LIN {X 0,Y 133.955,Z 458.167,A -85,B 0,C 180,E1 -24920.946,E2 -24920.946} C_VEL
LIN {X 0,Y 133.688,Z 459.441,A -85,B 0,C 180,E1 -24923.966,E2 -24923.966} C_VEL
LIN {X 0,Y 133.69,Z 460.263,A -85,B 0,C 180,E1 -24927.209,E2 -24927.209} C_VEL
LIN {X 0,Y 133.919,Z 460.549,A -85,B 0,C 180,E1 -24930.002,E2 -24930.002} C_VEL
LIN {X 0,Y 133.701,Z 460.227,A -85,B 0,C 180,E1 -24933.015,E2 -24933.015} C_VEL
LIN {X 0,Y 133.689,Z 459.406,A -85,B 0,C 180,E1 -24936.037,E2 -24936.037} C_VEL
LIN {X 0,Y 133.956,Z 458.108,A -85,B 0,C 180,E1 -24939.057,E2 -24939.057} C_VEL
LIN {X 0,Y 134.932,Z 455.141,A -85,B 0,C 180,E1 -24943.557,E2 -24943.557} C_VEL
LIN {X 0,Y 136.058,Z 452.45,A -85,B 0,C 180,E1 -24946.507,E2 -24946.507} C_VEL
LIN {X 0,Y 138.397,Z 447.21,A -85,B 0,C 180,E1 -24950.824,E2 -24950.824} C_VEL
LIN {X 0,Y 141.592,Z 440.318,A -85,B 0,C 180,E1 -24954.956,E2 -24954.956} C_VEL
LIN {X 0,Y 144.781,Z 432.803,A -85,B 0,C 180,E1 -24958.249,E2 -24958.249} C_VEL
LIN {X 0,Y 145.009,Z 432.247,A -85,B 0,C 180,E1 -24958.457,E2 -24958.457} C_VEL
LIN {X 0,Y 146.09,Z 428.19,A -85,B 0,C 180,E1 -24960.037,E2 -24960.037} C_VEL
LIN {X 0,Y 146.273,Z 421.026,A -85,B 0,C 180,E1 -24962.704,E2 -24962.704} C_VEL
LIN {X 0,Y 146.437,Z 413.294,A -85,B 0,C 180,E1 -24965.152,E2 -24965.152} C_VEL
LIN {X 0,Y 147.423,Z 408.136,A -85,B 0,C 180,E1 -24966.312,E2 -24966.312} C_VEL
LIN {X 0,Y 150.465,Z 396.447,A -85,B 0,C 180,E1 -24968.09,E2 -24968.09} C_VEL
LIN {X 0,Y 152.454,Z 386.113,A -85,B 0,C 180,E1 -24969.14,E2 -24969.14} C_VEL
LIN {X 0,Y 153.592,Z 376.297,A -85,B 0,C 180,E1 -24969.839,E2 -24969.839} C_VEL
LIN {X 0,Y 154.357,Z 363.434,A -85,B 0,C 180,E1 -24970.454,E2 -24970.454} C_VEL
LIN {X 0,Y 152.82,Z 343.881,A -85,B 0,C 180,E1 -24972.135,E2 -24972.135} C_VEL
LIN {X 0,Y 148.055,Z 331.746,A -85,B 0,C 180,E1 -24974.6,E2 -24974.6} C_VEL
LIN {X 0,Y 143.112,Z 321.493,A -85,B 0,C 180,E1 -24977.289,E2 -24977.289} C_VEL
LIN {X 0,Y 138.714,Z 313.265,A -85,B 0,C 180,E1 -24979.904,E2 -24979.904} C_VEL
LIN {X 0,Y 135.903,Z 309.235,A -85,B 0,C 180,E1 -24981.643,E2 -24981.643} C_VEL
LIN {X 0,Y 133.491,Z 306.239,A -85,B 0,C 180,E1 -24983.212,E2 -24983.212} C_VEL
LIN {X 0,Y 132.602,Z 304.57,A -85,B 0,C 180,E1 -24983.869,E2 -24983.869} C_VEL
LIN {X 0,Y 130.375,Z 302.63,A -85,B 0,C 180,E1 -24985.393,E2 -24985.393} C_VEL
LIN {X 0,Y 129.129,Z 300.08,A -85,B 0,C 180,E1 -24986.438,E2 -24986.438} C_VEL
LIN {X 0,Y 128.983,Z 299.233,A -85,B 0,C 180,E1 -24986.69,E2 -24986.69} C_VEL
LIN {X 0,Y 128.983,Z 299.231,A -85,B 0,C 180,E1 -24990.672,E2 -24990.672} C_VEL
LIN {X 0,Y 129.069,Z 299.222,A -85,B 0,C 180,E1 -24997.774,E2 -24997.774} C_VEL
LIN {X 0,Y 129.147,Z 299.205,A -85,B 0,C 180,E1 -25004.211,E2 -25004.211} C_VEL
LIN {X 0,Y 129.346,Z 299.177,A -85,B 0,C 180,E1 -25007.974,E2 -25007.974} C_VEL
LIN {X 0,Y 129.462,Z 299.131,A -85,B 0,C 180,E1 -25010.628,E2 -25010.628} C_VEL
LIN {X 0,Y 130.069,Z 299.082,A -85,B 0,C 180,E1 -25020,E2 -25020} C_VEL
LIN {X 0,Y 129.471,Z 299.171,A -85,B 0,C 180,E1 -25029.373,E2 -25029.373} C_VEL
LIN {X 0,Y 129.3,Z 299.165,A -85,B 0,C 180,E1 -25032.558,E2 -25032.558} C_VEL
LIN {X 0,Y 129.083,Z 299.212,A -85,B 0,C 180,E1 -25039.067,E2 -25039.067} C_VEL
LIN {X 0,Y 129.036,Z 299.216,A -85,B 0,C 180,E1 -25042.412,E2 -25042.412} C_VEL
LIN {X 0,Y 129.002,Z 299.223,A -85,B 0,C 180,E1 -25049.362,E2 -25049.362} C_VEL
LIN {X 0,Y 129.003,Z 299.198,A -85,B 0,C 180,E1 -25054.184,E2 -25054.184} C_VEL
LIN {X 0,Y 129.928,Z 301.964,A -85,B 0,C 180,E1 -25055.083,E2 -25055.083} C_VEL
LIN {X 0,Y 131.991,Z 304.22,A -85,B 0,C 180,E1 -25056.562,E2 -25056.562} C_VEL
LIN {X 0,Y 132.836,Z 304.916,A -85,B 0,C 180,E1 -25057.12,E2 -25057.12} C_VEL
LIN {X 0,Y 134.792,Z 308.132,A -85,B 0,C 180,E1 -25058.493,E2 -25058.493} C_VEL
LIN {X 0,Y 136.443,Z 309.987,A -85,B 0,C 180,E1 -25059.521,E2 -25059.521} C_VEL
LIN {X 0,Y 139.015,Z 313.601,A -85,B 0,C 180,E1 -25061.089,E2 -25061.089} C_VEL
LIN {X 0,Y 144.709,Z 322.224,A -85,B 0,C 180,E1 -25064.255,E2 -25064.255} C_VEL
LIN {X 0,Y 149.932,Z 331.119,A -85,B 0,C 180,E1 -25066.875,E2 -25066.875} C_VEL
LIN {X 0,Y 155.317,Z 341.866,A -85,B 0,C 180,E1 -25069.382,E2 -25069.382} C_VEL
LIN {X 0,Y 155.665,Z 342.647,A -85,B 0,C 180,E1 -25069.54,E2 -25069.54} C_VEL
LIN {X 0,Y 154.337,Z 363.927,A -85,B 0,C 180,E1 -25070.495,E2 -25070.495} C_VEL
LIN {X 0,Y 153.217,Z 374.014,A -85,B 0,C 180,E1 -25071.268,E2 -25071.268} C_VEL
LIN {X 0,Y 151.609,Z 384.894,A -85,B 0,C 180,E1 -25072.59,E2 -25072.59} C_VEL
LIN {X 0,Y 149.044,Z 395.291,A -85,B 0,C 180,E1 -25074.299,E2 -25074.299} C_VEL
LIN {X 0,Y 146.437,Z 403.647,A -85,B 0,C 180,E1 -25076.086,E2 -25076.086} C_VEL
LIN {X 0,Y 143.646,Z 411.532,A -85,B 0,C 180,E1 -25078.266,E2 -25078.266} C_VEL
LIN {X 0,Y 141.558,Z 417.18,A -85,B 0,C 180,E1 -25080.231,E2 -25080.231} C_VEL
LIN {X 0,Y 138.779,Z 423.499,A -85,B 0,C 180,E1 -25082.884,E2 -25082.884} C_VEL
LIN {X 0,Y 136.313,Z 428.747,A -85,B 0,C 180,E1 -25085.639,E2 -25085.639} C_VEL
LIN {X 0,Y 134.031,Z 433.13,A -85,B 0,C 180,E1 -25088.465,E2 -25088.465} C_VEL
LIN {X 0,Y 131.319,Z 438.275,A -85,B 0,C 180,E1 -25092.88,E2 -25092.88} C_VEL
LIN {X 0,Y 129.865,Z 440.911,A -85,B 0,C 180,E1 -25095.903,E2 -25095.903} C_VEL
LIN {X 0,Y 128.338,Z 443.792,A -85,B 0,C 180,E1 -25100.543,E2 -25100.543} C_VEL
LIN {X 0,Y 127.603,Z 445.049,A -85,B 0,C 180,E1 -25103.674,E2 -25103.674} C_VEL
LIN {X 0,Y 127.149,Z 445.841,A -85,B 0,C 180,E1 -25106.83,E2 -25106.83} C_VEL
LIN {X 0,Y 127.002,Z 446.143,A -85,B 0,C 180,E1 -25109.998,E2 -25109.998} C_VEL
LIN {X 0,Y 127.144,Z 445.862,A -85,B 0,C 180,E1 -25113.167,E2 -25113.167} C_VEL
LIN {X 0,Y 127.58,Z 445.113,A -85,B 0,C 180,E1 -25116.324,E2 -25116.324} C_VEL
LIN {X 0,Y 128.518,Z 443.539,A -85,B 0,C 180,E1 -25120.155,E2 -25120.155} C_VEL
LIN {X 0,Y 129.861,Z 441.06,A -85,B 0,C 180,E1 -25124.094,E2 -25124.094} C_VEL
LIN {X 0,Y 131.287,Z 438.472,A -85,B 0,C 180,E1 -25127.121,E2 -25127.121} C_VEL
LIN {X 0,Y 133.978,Z 433.382,A -85,B 0,C 180,E1 -25131.541,E2 -25131.541} C_VEL
LIN {X 0,Y 136.782,Z 427.897,A -85,B 0,C 180,E1 -25135.079,E2 -25135.079} C_VEL
LIN {X 0,Y 140.081,Z 420.989,A -85,B 0,C 180,E1 -25138.463,E2 -25138.463} C_VEL
LIN {X 0,Y 143.2,Z 413.068,A -85,B 0,C 180,E1 -25141.428,E2 -25141.428} C_VEL
LIN {X 0,Y 146.001,Z 405.5,A -85,B 0,C 180,E1 -25143.61,E2 -25143.61} C_VEL
LIN {X 0,Y 148.554,Z 397.558,A -85,B 0,C 180,E1 -25145.416,E2 -25145.416} C_VEL
LIN {X 0,Y 150.694,Z 389.348,A -85,B 0,C 180,E1 -25146.901,E2 -25146.901} C_VEL
LIN {X 0,Y 152.252,Z 381.809,A -85,B 0,C 180,E1 -25147.985,E2 -25147.985} C_VEL
LIN {X 0,Y 153.626,Z 372.764,A -85,B 0,C 180,E1 -25148.981,E2 -25148.981} C_VEL
LIN {X 0,Y 154.497,Z 363.901,A -85,B 0,C 180,E1 -25149.672,E2 -25149.672} C_VEL
LIN {X 0,Y 155.859,Z 342.918,A -85,B 0,C 180,E1 -25150.597,E2 -25150.597} C_VEL
LIN {X 0,Y 150.73,Z 332.485,A -85,B 0,C 180,E1 -25152.978,E2 -25152.978} C_VEL
LIN {X 0,Y 145.136,Z 322.922,A -85,B 0,C 180,E1 -25155.765,E2 -25155.765} C_VEL
LIN {X 0,Y 140.991,Z 316.577,A -85,B 0,C 180,E1 -25158.021,E2 -25158.021} C_VEL
LIN {X 0,Y 138.32,Z 312.726,A -85,B 0,C 180,E1 -25159.585,E2 -25159.585} C_VEL
LIN {X 0,Y 135.823,Z 309.153,A -85,B 0,C 180,E1 -25161.152,E2 -25161.152} C_VEL
LIN {X 0,Y 133.437,Z 306.163,A -85,B 0,C 180,E1 -25162.721,E2 -25162.721} C_VEL
LIN {X 0,Y 132.55,Z 304.531,A -85,B 0,C 180,E1 -25163.381,E2 -25163.381} C_VEL
LIN {X 0,Y 130.335,Z 302.594,A -85,B 0,C 180,E1 -25164.913,E2 -25164.913} C_VEL
LIN {X 0,Y 129.126,Z 299.874,A -85,B 0,C 180,E1 -25165.962,E2 -25165.962} C_VEL
LIN {X 0,Y 128.982,Z 299.226,A -85,B 0,C 180,E1 -25166.275,E2 -25166.275} C_VEL
LIN {X 0,Y 129.014,Z 299.225,A -85,B 0,C 180,E1 -25170.641,E2 -25170.641} C_VEL
LIN {X 0,Y 128.999,Z 299.227,A -85,B 0,C 180,E1 -25174.16,E2 -25174.16} C_VEL
LIN {X 0,Y 129.066,Z 299.213,A -85,B 0,C 180,E1 -25177.769,E2 -25177.769} C_VEL
LIN {X 0,Y 129.14,Z 299.174,A -85,B 0,C 180,E1 -25184.21,E2 -25184.21} C_VEL
LIN {X 0,Y 129.339,Z 299.165,A -85,B 0,C 180,E1 -25187.973,E2 -25187.973} C_VEL
LIN {X 0,Y 129.464,Z 299.171,A -85,B 0,C 180,E1 -25190.627,E2 -25190.627} C_VEL
LIN {X 0,Y 130.062,Z 299.084,A -85,B 0,C 180,E1 -25200,E2 -25200} C_VEL
LIN {X 0,Y 129.464,Z 299.164,A -85,B 0,C 180,E1 -25209.372,E2 -25209.372} C_VEL
LIN {X 0,Y 129.293,Z 299.19,A -85,B 0,C 180,E1 -25212.558,E2 -25212.558} C_VEL
LIN {X 0,Y 129.076,Z 299.217,A -85,B 0,C 180,E1 -25219.068,E2 -25219.068} C_VEL
LIN {X 0,Y 129.03,Z 299.227,A -85,B 0,C 180,E1 -25222.412,E2 -25222.412} C_VEL
LIN {X 0,Y 128.995,Z 299.233,A -85,B 0,C 180,E1 -25229.363,E2 -25229.363} C_VEL
LIN {X 0,Y 128.964,Z 299.27,A -85,B 0,C 180,E1 -25233.139,E2 -25233.139} C_VEL
LIN {X 0,Y 129.82,Z 301.8,A -85,B 0,C 180,E1 -25233.949,E2 -25233.949} C_VEL
LIN {X 0,Y 131.932,Z 304.15,A -85,B 0,C 180,E1 -25235.486,E2 -25235.486} C_VEL
LIN {X 0,Y 132.916,Z 305.054,A -85,B 0,C 180,E1 -25236.149,E2 -25236.149} C_VEL
LIN {X 0,Y 134.987,Z 308.332,A -85,B 0,C 180,E1 -25237.598,E2 -25237.598} C_VEL
LIN {X 0,Y 136.451,Z 309.935,A -85,B 0,C 180,E1 -25238.511,E2 -25238.511} C_VEL
LIN {X 0,Y 139.616,Z 314.845,A -85,B 0,C 180,E1 -25240.475,E2 -25240.475} C_VEL
LIN {X 0,Y 144.191,Z 323.442,A -85,B 0,C 180,E1 -25243.148,E2 -25243.148} C_VEL
LIN {X 0,Y 149.027,Z 333.816,A -85,B 0,C 180,E1 -25245.756,E2 -25245.756} C_VEL
LIN {X 0,Y 153.092,Z 344.587,A -85,B 0,C 180,E1 -25247.869,E2 -25247.869} C_VEL
LIN {X 0,Y 154.559,Z 365.309,A -85,B 0,C 180,E1 -25249.596,E2 -25249.596} C_VEL
LIN {X 0,Y 153.372,Z 380.616,A -85,B 0,C 180,E1 -25250.333,E2 -25250.333} C_VEL
LIN {X 0,Y 151.602,Z 391.787,A -85,B 0,C 180,E1 -25251.311,E2 -25251.311} C_VEL
LIN {X 0,Y 149.671,Z 400.473,A -85,B 0,C 180,E1 -25252.381,E2 -25252.381} C_VEL
LIN {X 0,Y 147.268,Z 409.143,A -85,B 0,C 180,E1 -25253.805,E2 -25253.805} C_VEL
LIN {X 0,Y 144.547,Z 417.44,A -85,B 0,C 180,E1 -25255.586,E2 -25255.586} C_VEL
LIN {X 0,Y 141.851,Z 424.645,A -85,B 0,C 180,E1 -25257.553,E2 -25257.553} C_VEL
LIN {X 0,Y 138.564,Z 432.657,A -85,B 0,C 180,E1 -25260.364,E2 -25260.364} C_VEL
LIN {X 0,Y 135.155,Z 440.129,A -85,B 0,C 180,E1 -25263.771,E2 -25263.771} C_VEL
LIN {X 0,Y 132.3,Z 445.995,A -85,B 0,C 180,E1 -25267.35,E2 -25267.35} C_VEL
LIN {X 0,Y 129.937,Z 450.626,A -85,B 0,C 180,E1 -25271.065,E2 -25271.065} C_VEL
LIN {X 0,Y 128.595,Z 453.651,A -85,B 0,C 180,E1 -25274.143,E2 -25274.143} C_VEL
LIN {X 0,Y 127.585,Z 456.005,A -85,B 0,C 180,E1 -25277.273,E2 -25277.273} C_VEL
LIN {X 0,Y 126.927,Z 457.774,A -85,B 0,C 180,E1 -25280.44,E2 -25280.44} C_VEL
LIN {X 0,Y 126.626,Z 459.049,A -85,B 0,C 180,E1 -25283.628,E2 -25283.628} C_VEL
LIN {X 0,Y 126.633,Z 459.91,A -85,B 0,C 180,E1 -25287.404,E2 -25287.404} C_VEL
LIN {X 0,Y 126.82,Z 460.157,A -85,B 0,C 180,E1 -25290.002,E2 -25290.002} C_VEL
LIN {X 0,Y 126.615,Z 459.835,A -85,B 0,C 180,E1 -25293.184,E2 -25293.184} C_VEL
LIN {X 0,Y 126.627,Z 459.013,A -85,B 0,C 180,E1 -25296.375,E2 -25296.375} C_VEL
LIN {X 0,Y 126.928,Z 457.715,A -85,B 0,C 180,E1 -25299.563,E2 -25299.563} C_VEL
LIN {X 0,Y 128.02,Z 454.747,A -85,B 0,C 180,E1 -25304.304,E2 -25304.304} C_VEL
LIN {X 0,Y 129.227,Z 452.054,A -85,B 0,C 180,E1 -25307.406,E2 -25307.406} C_VEL
LIN {X 0,Y 131.785,Z 446.817,A -85,B 0,C 180,E1 -25311.921,E2 -25311.921} C_VEL
LIN {X 0,Y 135.145,Z 439.921,A -85,B 0,C 180,E1 -25316.235,E2 -25316.235} C_VEL
LIN {X 0,Y 138.589,Z 432.366,A -85,B 0,C 180,E1 -25319.655,E2 -25319.655} C_VEL
LIN {X 0,Y 141.661,Z 425.004,A -85,B 0,C 180,E1 -25322.232,E2 -25322.232} C_VEL
LIN {X 0,Y 144.427,Z 417.444,A -85,B 0,C 180,E1 -25324.325,E2 -25324.325} C_VEL
LIN {X 0,Y 147.255,Z 408.695,A -85,B 0,C 180,E1 -25326.202,E2 -25326.202} C_VEL
LIN {X 0,Y 147.423,Z 408.136,A -85,B 0,C 180,E1 -25326.312,E2 -25326.312} C_VEL
LIN {X 0,Y 148.397,Z 402.979,A -85,B 0,C 180,E1 -25327.382,E2 -25327.382} C_VEL
LIN {X 0,Y 148.347,Z 394.3,A -85,B 0,C 180,E1 -25329.252,E2 -25329.252} C_VEL
LIN {X 0,Y 147.785,Z 385.247,A -85,B 0,C 180,E1 -25330.819,E2 -25330.819} C_VEL
LIN {X 0,Y 147.904,Z 379.504,A -85,B 0,C 180,E1 -25331.386,E2 -25331.386} C_VEL
LIN {X 0,Y 148.981,Z 364.614,A -85,B 0,C 180,E1 -25332.14,E2 -25332.14} C_VEL
LIN {X 0,Y 147.735,Z 346.63,A -85,B 0,C 180,E1 -25333.739,E2 -25333.739} C_VEL
LIN {X 0,Y 143.311,Z 335.144,A -85,B 0,C 180,E1 -25336.234,E2 -25336.234} C_VEL
LIN {X 0,Y 138.463,Z 324.854,A -85,B 0,C 180,E1 -25339.125,E2 -25339.125} C_VEL
LIN {X 0,Y 134.783,Z 318.011,A -85,B 0,C 180,E1 -25341.505,E2 -25341.505} C_VEL
LIN {X 0,Y 132.341,Z 314.562,A -85,B 0,C 180,E1 -25343.136,E2 -25343.136} C_VEL
LIN {X 0,Y 130.013,Z 311.221,A -85,B 0,C 180,E1 -25344.815,E2 -25344.815} C_VEL
LIN {X 0,Y 126.908,Z 307.447,A -85,B 0,C 180,E1 -25347.203,E2 -25347.203} C_VEL
LIN {X 0,Y 126.017,Z 305.712,A -85,B 0,C 180,E1 -25348.007,E2 -25348.007} C_VEL
LIN {X 0,Y 123.536,Z 303.83,A -85,B 0,C 180,E1 -25350.079,E2 -25350.079} C_VEL
LIN {X 0,Y 122.11,Z 301.179,A -85,B 0,C 180,E1 -25351.559,E2 -25351.559} C_VEL
LIN {X 0,Y 121.88,Z 300.112,A -85,B 0,C 180,E1 -25351.942,E2 -25351.942} C_VEL
LIN {X 0,Y 121.981,Z 300.104,A -85,B 0,C 180,E1 -25357.202,E2 -25357.202} C_VEL
LIN {X 0,Y 122.06,Z 300.089,A -85,B 0,C 180,E1 -25363.269,E2 -25363.269} C_VEL
LIN {X 0,Y 122.289,Z 300.058,A -85,B 0,C 180,E1 -25367.694,E2 -25367.694} C_VEL
LIN {X 0,Y 122.391,Z 300.014,A -85,B 0,C 180,E1 -25370.081,E2 -25370.081} C_VEL
LIN {X 0,Y 122.558,Z 300.027,A -85,B 0,C 180,E1 -25376.713,E2 -25376.713} C_VEL
LIN {X 0,Y 123.022,Z 299.958,A -85,B 0,C 180,E1 -25380,E2 -25380} C_VEL
LIN {X 0,Y 122.391,Z 300.026,A -85,B 0,C 180,E1 -25386.889,E2 -25386.889} C_VEL
LIN {X 0,Y 122.29,Z 300.039,A -85,B 0,C 180,E1 -25392.308,E2 -25392.308} C_VEL
LIN {X 0,Y 122.06,Z 300.056,A -85,B 0,C 180,E1 -25396.732,E2 -25396.732} C_VEL
LIN {X 0,Y 121.981,Z 300.094,A -85,B 0,C 180,E1 -25402.799,E2 -25402.799} C_VEL
LIN {X 0,Y 121.959,Z 300.136,A -85,B 0,C 180,E1 -25409.009,E2 -25409.009} C_VEL
LIN {X 0,Y 122.813,Z 302.78,A -85,B 0,C 180,E1 -25410.039,E2 -25410.039} C_VEL
LIN {X 0,Y 124.819,Z 305.005,A -85,B 0,C 180,E1 -25411.862,E2 -25411.862} C_VEL
LIN {X 0,Y 126.222,Z 306.072,A -85,B 0,C 180,E1 -25412.999,E2 -25412.999} C_VEL
LIN {X 0,Y 128.002,Z 309.087,A -85,B 0,C 180,E1 -25414.521,E2 -25414.521} C_VEL
LIN {X 0,Y 129.971,Z 311.162,A -85,B 0,C 180,E1 -25415.975,E2 -25415.975} C_VEL
LIN {X 0,Y 132.546,Z 314.779,A -85,B 0,C 180,E1 -25417.822,E2 -25417.822} C_VEL
LIN {X 0,Y 138.419,Z 323.322,A -85,B 0,C 180,E1 -25421.558,E2 -25421.558} C_VEL
LIN {X 0,Y 144.642,Z 333.733,A -85,B 0,C 180,E1 -25425.03,E2 -25425.03} C_VEL
LIN {X 0,Y 150.226,Z 344.979,A -85,B 0,C 180,E1 -25427.868,E2 -25427.868} C_VEL
LIN {X 0,Y 148.944,Z 364.375,A -85,B 0,C 180,E1 -25428.766,E2 -25428.766} C_VEL
LIN {X 0,Y 147.653,Z 375.081,A -85,B 0,C 180,E1 -25429.603,E2 -25429.603} C_VEL
LIN {X 0,Y 145.627,Z 386.917,A -85,B 0,C 180,E1 -25431.141,E2 -25431.141} C_VEL
LIN {X 0,Y 143.358,Z 395.687,A -85,B 0,C 180,E1 -25432.649,E2 -25432.649} C_VEL
LIN {X 0,Y 140.613,Z 404.043,A -85,B 0,C 180,E1 -25434.475,E2 -25434.475} C_VEL
LIN {X 0,Y 137.69,Z 411.925,A -85,B 0,C 180,E1 -25436.72,E2 -25436.72} C_VEL
LIN {X 0,Y 134.71,Z 419.265,A -85,B 0,C 180,E1 -25439.423,E2 -25439.423} C_VEL
LIN {X 0,Y 131.145,Z 426.708,A -85,B 0,C 180,E1 -25442.901,E2 -25442.901} C_VEL
LIN {X 0,Y 127.481,Z 433.522,A -85,B 0,C 180,E1 -25447.298,E2 -25447.298} C_VEL
LIN {X 0,Y 124.567,Z 438.667,A -85,B 0,C 180,E1 -25451.921,E2 -25451.921} C_VEL
LIN {X 0,Y 123.02,Z 441.303,A -85,B 0,C 180,E1 -25455.101,E2 -25455.101} C_VEL
LIN {X 0,Y 121.363,Z 444.183,A -85,B 0,C 180,E1 -25459.994,E2 -25459.994} C_VEL
LIN {X 0,Y 120.56,Z 445.441,A -85,B 0,C 180,E1 -25463.303,E2 -25463.303} C_VEL
LIN {X 0,Y 120.09,Z 446.232,A -85,B 0,C 180,E1 -25466.643,E2 -25466.643} C_VEL
LIN {X 0,Y 119.931,Z 446.533,A -85,B 0,C 180,E1 -25469.998,E2 -25469.998} C_VEL
LIN {X 0,Y 120.084,Z 446.253,A -85,B 0,C 180,E1 -25473.353,E2 -25473.353} C_VEL
LIN {X 0,Y 120.555,Z 445.503,A -85,B 0,C 180,E1 -25476.694,E2 -25476.694} C_VEL
LIN {X 0,Y 121.322,Z 444.289,A -85,B 0,C 180,E1 -25480.006,E2 -25480.006} C_VEL
LIN {X 0,Y 123.017,Z 441.45,A -85,B 0,C 180,E1 -25484.895,E2 -25484.895} C_VEL
LIN {X 0,Y 124.526,Z 438.863,A -85,B 0,C 180,E1 -25488.082,E2 -25488.082} C_VEL
LIN {X 0,Y 127.427,Z 433.771,A -85,B 0,C 180,E1 -25492.708,E2 -25492.708} C_VEL
LIN {X 0,Y 130.4,Z 428.286,A -85,B 0,C 180,E1 -25496.398,E2 -25496.398} C_VEL
LIN {X 0,Y 133.904,Z 421.377,A -85,B 0,C 180,E1 -25499.906,E2 -25499.906} C_VEL
LIN {X 0,Y 137.221,Z 413.455,A -85,B 0,C 180,E1 -25502.966,E2 -25502.966} C_VEL
LIN {X 0,Y 140.156,Z 405.887,A -85,B 0,C 180,E1 -25505.214,E2 -25505.214} C_VEL
LIN {X 0,Y 142.855,Z 397.943,A -85,B 0,C 180,E1 -25507.058,E2 -25507.058} C_VEL
LIN {X 0,Y 145.092,Z 389.733,A -85,B 0,C 180,E1 -25508.581,E2 -25508.581} C_VEL
LIN {X 0,Y 147.029,Z 380.751,A -85,B 0,C 180,E1 -25509.858,E2 -25509.858} C_VEL
LIN {X 0,Y 148.428,Z 371.27,A -85,B 0,C 180,E1 -25510.877,E2 -25510.877} C_VEL
LIN {X 0,Y 149.468,Z 360.824,A -85,B 0,C 180,E1 -25511.589,E2 -25511.589} C_VEL
LIN {X 0,Y 150.43,Z 345.249,A -85,B 0,C 180,E1 -25512.269,E2 -25512.269} C_VEL
LIN {X 0,Y 145.035,Z 334.384,A -85,B 0,C 180,E1 -25515.009,E2 -25515.009} C_VEL
LIN {X 0,Y 139.531,Z 325.12,A -85,B 0,C 180,E1 -25518.047,E2 -25518.047} C_VEL
LIN {X 0,Y 134.959,Z 318.208,A -85,B 0,C 180,E1 -25520.855,E2 -25520.855} C_VEL
LIN {X 0,Y 132.401,Z 314.611,A -85,B 0,C 180,E1 -25522.571,E2 -25522.571} C_VEL
LIN {X 0,Y 129.875,Z 310.919,A -85,B 0,C 180,E1 -25524.418,E2 -25524.418} C_VEL
LIN {X 0,Y 127.202,Z 307.944,A -85,B 0,C 180,E1 -25526.46,E2 -25526.46} C_VEL
LIN {X 0,Y 126.013,Z 305.69,A -85,B 0,C 180,E1 -25527.533,E2 -25527.533} C_VEL
LIN {X 0,Y 123.603,Z 303.9,A -85,B 0,C 180,E1 -25529.564,E2 -25529.564} C_VEL
LIN {X 0,Y 122.245,Z 301.395,A -85,B 0,C 180,E1 -25530.98,E2 -25530.98} C_VEL
LIN {X 0,Y 121.928,Z 300.101,A -85,B 0,C 180,E1 -25531.498,E2 -25531.498} C_VEL
LIN {X 0,Y 121.984,Z 300.094,A -85,B 0,C 180,E1 -25537.189,E2 -25537.189} C_VEL
LIN {X 0,Y 122.055,Z 300.061,A -85,B 0,C 180,E1 -25543.267,E2 -25543.267} C_VEL
LIN {X 0,Y 122.283,Z 300.038,A -85,B 0,C 180,E1 -25547.691,E2 -25547.691} C_VEL
LIN {X 0,Y 122.39,Z 300.051,A -85,B 0,C 180,E1 -25550.08,E2 -25550.08} C_VEL
LIN {X 0,Y 122.551,Z 299.988,A -85,B 0,C 180,E1 -25556.712,E2 -25556.712} C_VEL
LIN {X 0,Y 123.015,Z 299.961,A -85,B 0,C 180,E1 -25560,E2 -25560} C_VEL
LIN {X 0,Y 122.404,Z 300.046,A -85,B 0,C 180,E1 -25566.594,E2 -25566.594} C_VEL
LIN {X 0,Y 122.391,Z 300.042,A -85,B 0,C 180,E1 -25569.919,E2 -25569.919} C_VEL
LIN {X 0,Y 122.182,Z 300.078,A -85,B 0,C 180,E1 -25573.302,E2 -25573.302} C_VEL
LIN {X 0,Y 121.981,Z 300.097,A -85,B 0,C 180,E1 -25580.224,E2 -25580.224} C_VEL
LIN {X 0,Y 121.907,Z 300.109,A -85,B 0,C 180,E1 -25583.8,E2 -25583.8} C_VEL
LIN {X 0,Y 121.896,Z 300.161,A -85,B 0,C 180,E1 -25587.836,E2 -25587.836} C_VEL
LIN {X 0,Y 122.59,Z 302.371,A -85,B 0,C 180,E1 -25588.697,E2 -25588.697} C_VEL
LIN {X 0,Y 124.523,Z 304.801,A -85,B 0,C 180,E1 -25590.527,E2 -25590.527} C_VEL
LIN {X 0,Y 126.229,Z 306.082,A -85,B 0,C 180,E1 -25591.932,E2 -25591.932} C_VEL
LIN {X 0,Y 128.297,Z 309.395,A -85,B 0,C 180,E1 -25593.691,E2 -25593.691} C_VEL
LIN {X 0,Y 130.005,Z 311.16,A -85,B 0,C 180,E1 -25594.954,E2 -25594.954} C_VEL
LIN {X 0,Y 132.549,Z 314.771,A -85,B 0,C 180,E1 -25596.797,E2 -25596.797} C_VEL
LIN {X 0,Y 135.721,Z 319.451,A -85,B 0,C 180,E1 -25598.913,E2 -25598.913} C_VEL
LIN {X 0,Y 140.916,Z 329.78,A -85,B 0,C 180,E1 -25602.197,E2 -25602.197} C_VEL
LIN {X 0,Y 144.887,Z 338.802,A -85,B 0,C 180,E1 -25604.505,E2 -25604.505} C_VEL
LIN {X 0,Y 148.019,Z 347.59,A -85,B 0,C 180,E1 -25606.287,E2 -25606.287} C_VEL
LIN {X 0,Y 149.171,Z 365.627,A -85,B 0,C 180,E1 -25607.854,E2 -25607.854} C_VEL
LIN {X 0,Y 147.883,Z 380.953,A -85,B 0,C 180,E1 -25608.629,E2 -25608.629} C_VEL
LIN {X 0,Y 146.254,Z 390.916,A -85,B 0,C 180,E1 -25609.521,E2 -25609.521} C_VEL
LIN {X 0,Y 144.112,Z 400.087,A -85,B 0,C 180,E1 -25610.658,E2 -25610.658} C_VEL
LIN {X 0,Y 141.591,Z 408.755,A -85,B 0,C 180,E1 -25612.105,E2 -25612.105} C_VEL
LIN {X 0,Y 138.75,Z 417.052,A -85,B 0,C 180,E1 -25613.929,E2 -25613.929} C_VEL
LIN {X 0,Y 135.899,Z 424.256,A -85,B 0,C 180,E1 -25615.944,E2 -25615.944} C_VEL
LIN {X 0,Y 133.211,Z 430.555,A -85,B 0,C 180,E1 -25618.16,E2 -25618.16} C_VEL
LIN {X 0,Y 130.14,Z 436.89,A -85,B 0,C 180,E1 -25620.922,E2 -25620.922} C_VEL
LIN {X 0,Y 127.537,Z 442.167,A -85,B 0,C 180,E1 -25623.844,E2 -25623.844} C_VEL
LIN {X 0,Y 125.2,Z 446.568,A -85,B 0,C 180,E1 -25626.864,E2 -25626.864} C_VEL
LIN {X 0,Y 122.442,Z 451.773,A -85,B 0,C 180,E1 -25631.599,E2 -25631.599} C_VEL
LIN {X 0,Y 120.632,Z 455.611,A -85,B 0,C 180,E1 -25636.526,E2 -25636.526} C_VEL
LIN {X 0,Y 119.925,Z 457.383,A -85,B 0,C 180,E1 -25639.876,E2 -25639.876} C_VEL
LIN {X 0,Y 119.56,Z 458.657,A -85,B 0,C 180,E1 -25643.25,E2 -25643.25} C_VEL
LIN {X 0,Y 119.565,Z 459.573,A -85,B 0,C 180,E1 -25647.783,E2 -25647.783} C_VEL
LIN {X 0,Y 119.724,Z 459.766,A -85,B 0,C 180,E1 -25650.002,E2 -25650.002} C_VEL
LIN {X 0,Y 119.53,Z 459.443,A -85,B 0,C 180,E1 -25653.372,E2 -25653.372} C_VEL
LIN {X 0,Y 119.561,Z 458.62,A -85,B 0,C 180,E1 -25656.753,E2 -25656.753} C_VEL
LIN {X 0,Y 119.925,Z 457.322,A -85,B 0,C 180,E1 -25660.127,E2 -25660.127} C_VEL
LIN {X 0,Y 121.142,Z 454.353,A -85,B 0,C 180,E1 -25665.135,E2 -25665.135} C_VEL
LIN {X 0,Y 122.441,Z 451.659,A -85,B 0,C 180,E1 -25668.404,E2 -25668.404} C_VEL
LIN {X 0,Y 125.198,Z 446.421,A -85,B 0,C 180,E1 -25673.14,E2 -25673.14} C_VEL
LIN {X 0,Y 128.766,Z 439.524,A -85,B 0,C 180,E1 -25677.642,E2 -25677.642} C_VEL
LIN {X 0,Y 132.432,Z 432.013,A -85,B 0,C 180,E1 -25681.161,E2 -25681.161} C_VEL
LIN {X 0,Y 135.699,Z 424.546,A -85,B 0,C 180,E1 -25683.86,E2 -25683.86} C_VEL
LIN {X 0,Y 138.605,Z 417.047,A -85,B 0,C 180,E1 -25685.985,E2 -25685.985} C_VEL
LIN {X 0,Y 141.577,Z 408.298,A -85,B 0,C 180,E1 -25687.903,E2 -25687.903} C_VEL
LIN {X 0,Y 144.484,Z 398.024,A -85,B 0,C 180,E1 -25689.578,E2 -25689.578} C_VEL
LIN {X 0,Y 146.859,Z 386.769,A -85,B 0,C 180,E1 -25690.795,E2 -25690.795} C_VEL
LIN {X 0,Y 147.904,Z 379.504,A -85,B 0,C 180,E1 -25691.386,E2 -25691.386} C_VEL
LIN {X 0,Y 147.734,Z 375.689,A -85,B 0,C 180,E1 -25691.778,E2 -25691.778} C_VEL
LIN {X 0,Y 146.08,Z 369.808,A -85,B 0,C 180,E1 -25692.823,E2 -25692.823} C_VEL
LIN {X 0,Y 143.792,Z 362.747,A -85,B 0,C 180,E1 -25694.141,E2 -25694.141} C_VEL
LIN {X 0,Y 143.42,Z 360.197,A -85,B 0,C 180,E1 -25694.454,E2 -25694.454} C_VEL
LIN {X 0,Y 142.64,Z 349.116,A -85,B 0,C 180,E1 -25695.527,E2 -25695.527} C_VEL
LIN {X 0,Y 138.633,Z 338.403,A -85,B 0,C 180,E1 -25698.015,E2 -25698.015} C_VEL
LIN {X 0,Y 133.598,Z 327.483,A -85,B 0,C 180,E1 -25701.341,E2 -25701.341} C_VEL
LIN {X 0,Y 131.174,Z 323.051,A -85,B 0,C 180,E1 -25703.054,E2 -25703.054} C_VEL
LIN {X 0,Y 128.986,Z 319.915,A -85,B 0,C 180,E1 -25704.638,E2 -25704.638} C_VEL
LIN {X 0,Y 126.369,Z 316.216,A -85,B 0,C 180,E1 -25706.688,E2 -25706.688} C_VEL
LIN {X 0,Y 123.879,Z 312.802,A -85,B 0,C 180,E1 -25708.823,E2 -25708.823} C_VEL
LIN {X 0,Y 123.182,Z 311.874,A -85,B 0,C 180,E1 -25709.457,E2 -25709.457} C_VEL
LIN {X 0,Y 120.7,Z 309.314,A -85,B 0,C 180,E1 -25711.792,E2 -25711.792} C_VEL
LIN {X 0,Y 119.361,Z 306.746,A -85,B 0,C 180,E1 -25713.323,E2 -25713.323} C_VEL
LIN {X 0,Y 116.939,Z 305.194,A -85,B 0,C 180,E1 -25715.968,E2 -25715.968} C_VEL
LIN {X 0,Y 115.24,Z 302.41,A -85,B 0,C 180,E1 -25718.347,E2 -25718.347} C_VEL
LIN {X 0,Y 114.935,Z 300.977,A -85,B 0,C 180,E1 -25719.064,E2 -25719.064} C_VEL
LIN {X 0,Y 115.081,Z 300.962,A -85,B 0,C 180,E1 -25725.861,E2 -25725.861} C_VEL
LIN {X 0,Y 115.307,Z 300.901,A -85,B 0,C 180,E1 -25729.464,E2 -25729.464} C_VEL
LIN {X 0,Y 115.485,Z 300.905,A -85,B 0,C 180,E1 -25736.511,E2 -25736.511} C_VEL
LIN {X 0,Y 115.95,Z 300.837,A -85,B 0,C 180,E1 -25740,E2 -25740} C_VEL
LIN {X 0,Y 115.351,Z 300.905,A -85,B 0,C 180,E1 -25746.999,E2 -25746.999} C_VEL
LIN {X 0,Y 115.207,Z 300.916,A -85,B 0,C 180,E1 -25752.557,E2 -25752.557} C_VEL
LIN {X 0,Y 114.965,Z 300.948,A -85,B 0,C 180,E1 -25757.798,E2 -25757.798} C_VEL
LIN {X 0,Y 114.948,Z 301.145,A -85,B 0,C 180,E1 -25761.902,E2 -25761.902} C_VEL
LIN {X 0,Y 115.768,Z 303.607,A -85,B 0,C 180,E1 -25763.298,E2 -25763.298} C_VEL
LIN {X 0,Y 117.627,Z 305.827,A -85,B 0,C 180,E1 -25765.67,E2 -25765.67} C_VEL
LIN {X 0,Y 119.541,Z 306.998,A -85,B 0,C 180,E1 -25767.699,E2 -25767.699} C_VEL
LIN {X 0,Y 121.193,Z 309.986,A -85,B 0,C 180,E1 -25769.535,E2 -25769.535} C_VEL
LIN {X 0,Y 123.599,Z 312.317,A -85,B 0,C 180,E1 -25771.734,E2 -25771.734} C_VEL
LIN {X 0,Y 126.052,Z 315.92,A -85,B 0,C 180,E1 -25773.887,E2 -25773.887} C_VEL
LIN {X 0,Y 127.297,Z 317.475,A -85,B 0,C 180,E1 -25774.877,E2 -25774.877} C_VEL
LIN {X 0,Y 130.877,Z 322.682,A -85,B 0,C 180,E1 -25777.564,E2 -25777.564} C_VEL
LIN {X 0,Y 135.247,Z 329.262,A -85,B 0,C 180,E1 -25780.478,E2 -25780.478} C_VEL
LIN {X 0,Y 141.116,Z 339.48,A -85,B 0,C 180,E1 -25783.978,E2 -25783.978} C_VEL
LIN {X 0,Y 144.861,Z 347.157,A -85,B 0,C 180,E1 -25786.037,E2 -25786.037} C_VEL
LIN {X 0,Y 143.672,Z 365.156,A -85,B 0,C 180,E1 -25786.931,E2 -25786.931} C_VEL
LIN {X 0,Y 142.288,Z 375.959,A -85,B 0,C 180,E1 -25787.808,E2 -25787.808} C_VEL
LIN {X 0,Y 140.189,Z 387.313,A -85,B 0,C 180,E1 -25789.327,E2 -25789.327} C_VEL
LIN {X 0,Y 137.799,Z 396.082,A -85,B 0,C 180,E1 -25790.863,E2 -25790.863} C_VEL
LIN {X 0,Y 134.926,Z 404.437,A -85,B 0,C 180,E1 -25792.732,E2 -25792.732} C_VEL
LIN {X 0,Y 131.843,Z 412.319,A -85,B 0,C 180,E1 -25795.036,E2 -25795.036} C_VEL
LIN {X 0,Y 128.674,Z 419.658,A -85,B 0,C 180,E1 -25797.822,E2 -25797.822} C_VEL
LIN {X 0,Y 124.893,Z 427.101,A -85,B 0,C 180,E1 -25801.423,E2 -25801.423} C_VEL
LIN {X 0,Y 120.995,Z 433.914,A -85,B 0,C 180,E1 -25806.007,E2 -25806.007} C_VEL
LIN {X 0,Y 117.846,Z 439.06,A -85,B 0,C 180,E1 -25810.851,E2 -25810.851} C_VEL
LIN {X 0,Y 116.185,Z 441.695,A -85,B 0,C 180,E1 -25814.203,E2 -25814.203} C_VEL
LIN {X 0,Y 114.409,Z 444.574,A -85,B 0,C 180,E1 -25819.379,E2 -25819.379} C_VEL
LIN {X 0,Y 113.521,Z 445.833,A -85,B 0,C 180,E1 -25822.886,E2 -25822.886} C_VEL
LIN {X 0,Y 113.014,Z 446.623,A -85,B 0,C 180,E1 -25826.433,E2 -25826.433} C_VEL
LIN {X 0,Y 112.842,Z 446.924,A -85,B 0,C 180,E1 -25829.998,E2 -25829.998} C_VEL
LIN {X 0,Y 113.009,Z 446.644,A -85,B 0,C 180,E1 -25833.564,E2 -25833.564} C_VEL
LIN {X 0,Y 114.183,Z 444.965,A -85,B 0,C 180,E1 -25839.999,E2 -25839.999} C_VEL
LIN {X 0,Y 115.531,Z 442.977,A -85,B 0,C 180,E1 -25844.081,E2 -25844.081} C_VEL
LIN {X 0,Y 117.817,Z 439.252,A -85,B 0,C 180,E1 -25849.151,E2 -25849.151} C_VEL
LIN {X 0,Y 120.94,Z 434.159,A -85,B 0,C 180,E1 -25854.001,E2 -25854.001} C_VEL
LIN {X 0,Y 124.102,Z 428.675,A -85,B 0,C 180,E1 -25857.851,E2 -25857.851} C_VEL
LIN {X 0,Y 127.824,Z 421.765,A -85,B 0,C 180,E1 -25861.486,E2 -25861.486} C_VEL
LIN {X 0,Y 131.345,Z 413.842,A -85,B 0,C 180,E1 -25864.645,E2 -25864.645} C_VEL
LIN {X 0,Y 134.446,Z 406.273,A -85,B 0,C 180,E1 -25866.95,E2 -25866.95} C_VEL
LIN {X 0,Y 137.284,Z 398.328,A -85,B 0,C 180,E1 -25868.835,E2 -25868.835} C_VEL
LIN {X 0,Y 139.634,Z 390.117,A -85,B 0,C 180,E1 -25870.39,E2 -25870.39} C_VEL
LIN {X 0,Y 141.547,Z 381.691,A -85,B 0,C 180,E1 -25871.627,E2 -25871.627} C_VEL
LIN {X 0,Y 143.059,Z 372.284,A -85,B 0,C 180,E1 -25872.674,E2 -25872.674} C_VEL
LIN {X 0,Y 144.154,Z 362.075,A -85,B 0,C 180,E1 -25873.411,E2 -25873.411} C_VEL
LIN {X 0,Y 145.103,Z 347.554,A -85,B 0,C 180,E1 -25874.081,E2 -25874.081} C_VEL
LIN {X 0,Y 139.9,Z 337.191,A -85,B 0,C 180,E1 -25876.974,E2 -25876.974} C_VEL
LIN {X 0,Y 134.512,Z 327.997,A -85,B 0,C 180,E1 -25880.279,E2 -25880.279} C_VEL
LIN {X 0,Y 129.55,Z 320.545,A -85,B 0,C 180,E1 -25883.721,E2 -25883.721} C_VEL
LIN {X 0,Y 126.472,Z 316.291,A -85,B 0,C 180,E1 -25886.12,E2 -25886.12} C_VEL
LIN {X 0,Y 123.899,Z 312.838,A -85,B 0,C 180,E1 -25888.336,E2 -25888.336} C_VEL
LIN {X 0,Y 123.094,Z 311.764,A -85,B 0,C 180,E1 -25889.079,E2 -25889.079} C_VEL
LIN {X 0,Y 120.725,Z 309.331,A -85,B 0,C 180,E1 -25891.339,E2 -25891.339} C_VEL
LIN {X 0,Y 119.416,Z 306.759,A -85,B 0,C 180,E1 -25892.863,E2 -25892.863} C_VEL
LIN {X 0,Y 116.8,Z 305.022,A -85,B 0,C 180,E1 -25895.787,E2 -25895.787} C_VEL
LIN {X 0,Y 115.184,Z 302.228,A -85,B 0,C 180,E1 -25898.139,E2 -25898.139} C_VEL
LIN {X 0,Y 114.91,Z 300.979,A -85,B 0,C 180,E1 -25898.706,E2 -25898.706} C_VEL
LIN {X 0,Y 115.075,Z 300.922,A -85,B 0,C 180,E1 -25905.86,E2 -25905.86} C_VEL
LIN {X 0,Y 115.304,Z 300.929,A -85,B 0,C 180,E1 -25909.463,E2 -25909.463} C_VEL
LIN {X 0,Y 115.477,Z 300.867,A -85,B 0,C 180,E1 -25916.51,E2 -25916.51} C_VEL
LIN {X 0,Y 115.967,Z 300.836,A -85,B 0,C 180,E1 -25920,E2 -25920} C_VEL
LIN {X 0,Y 115.346,Z 300.927,A -85,B 0,C 180,E1 -25926.999,E2 -25926.999} C_VEL
LIN {X 0,Y 115.199,Z 300.945,A -85,B 0,C 180,E1 -25932.557,E2 -25932.557} C_VEL
LIN {X 0,Y 114.924,Z 300.981,A -85,B 0,C 180,E1 -25940.587,E2 -25940.587} C_VEL
LIN {X 0,Y 115.627,Z 303.334,A -85,B 0,C 180,E1 -25941.86,E2 -25941.86} C_VEL
LIN {X 0,Y 117.797,Z 305.94,A -85,B 0,C 180,E1 -25944.685,E2 -25944.685} C_VEL
LIN {X 0,Y 119.51,Z 306.978,A -85,B 0,C 180,E1 -25946.523,E2 -25946.523} C_VEL
LIN {X 0,Y 121.405,Z 310.236,A -85,B 0,C 180,E1 -25948.629,E2 -25948.629} C_VEL
LIN {X 0,Y 123.715,Z 312.447,A -85,B 0,C 180,E1 -25950.748,E2 -25950.748} C_VEL
LIN {X 0,Y 126.264,Z 316.094,A -85,B 0,C 180,E1 -25952.986,E2 -25952.986} C_VEL
LIN {X 0,Y 127.401,Z 317.564,A -85,B 0,C 180,E1 -25953.899,E2 -25953.899} C_VEL
LIN {X 0,Y 130.802,Z 322.448,A -85,B 0,C 180,E1 -25956.469,E2 -25956.469} C_VEL
LIN {X 0,Y 132.753,Z 325.754,A -85,B 0,C 180,E1 -25957.863,E2 -25957.863} C_VEL
LIN {X 0,Y 137.82,Z 336.297,A -85,B 0,C 180,E1 -25961.279,E2 -25961.279} C_VEL
LIN {X 0,Y 142.078,Z 347.187,A -85,B 0,C 180,E1 -25963.953,E2 -25963.953} C_VEL
LIN {X 0,Y 142.937,Z 349.704,A -85,B 0,C 180,E1 -25964.48,E2 -25964.48} C_VEL
LIN {X 0,Y 143.898,Z 366.473,A -85,B 0,C 180,E1 -25966.007,E2 -25966.007} C_VEL
LIN {X 0,Y 142.537,Z 381.175,A -85,B 0,C 180,E1 -25966.793,E2 -25966.793} C_VEL
LIN {X 0,Y 140.799,Z 391.081,A -85,B 0,C 180,E1 -25967.709,E2 -25967.709} C_VEL
LIN {X 0,Y 138.7,Z 399.702,A -85,B 0,C 180,E1 -25968.8,E2 -25968.8} C_VEL
LIN {X 0,Y 136.073,Z 408.368,A -85,B 0,C 180,E1 -25970.274,E2 -25970.274} C_VEL
LIN {X 0,Y 133.088,Z 416.66,A -85,B 0,C 180,E1 -25972.131,E2 -25972.131} C_VEL
LIN {X 0,Y 129.881,Z 424.303,A -85,B 0,C 180,E1 -25974.333,E2 -25974.333} C_VEL
LIN {X 0,Y 127.218,Z 430.164,A -85,B 0,C 180,E1 -25976.468,E2 -25976.468} C_VEL
LIN {X 0,Y 123.983,Z 436.5,A -85,B 0,C 180,E1 -25979.327,E2 -25979.327} C_VEL
LIN {X 0,Y 121.179,Z 441.775,A -85,B 0,C 180,E1 -25982.358,E2 -25982.358} C_VEL
LIN {X 0,Y 118.676,Z 446.176,A -85,B 0,C 180,E1 -25985.512,E2 -25985.512} C_VEL
LIN {X 0,Y 115.683,Z 451.38,A -85,B 0,C 180,E1 -25990.482,E2 -25990.482} C_VEL
LIN {X 0,Y 113.718,Z 455.219,A -85,B 0,C 180,E1 -25995.69,E2 -25995.69} C_VEL
LIN {X 0,Y 112.918,Z 456.99,A -85,B 0,C 180,E1 -25999.241,E2 -25999.241} C_VEL
LIN {X 0,Y 112.492,Z 458.264,A -85,B 0,C 180,E1 -26002.824,E2 -26002.824} C_VEL
LIN {X 0,Y 112.496,Z 459.245,A -85,B 0,C 180,E1 -26008.317,E2 -26008.317} C_VEL
LIN {X 0,Y 112.625,Z 459.374,A -85,B 0,C 180,E1 -26010.002,E2 -26010.002} C_VEL
LIN {X 0,Y 112.43,Z 459.05,A -85,B 0,C 180,E1 -26013.586,E2 -26013.586} C_VEL
LIN {X 0,Y 112.493,Z 458.227,A -85,B 0,C 180,E1 -26017.18,E2 -26017.18} C_VEL
LIN {X 0,Y 112.918,Z 456.928,A -85,B 0,C 180,E1 -26020.763,E2 -26020.763} C_VEL
LIN {X 0,Y 114.278,Z 453.959,A -85,B 0,C 180,E1 -26026.068,E2 -26026.068} C_VEL
LIN {X 0,Y 115.683,Z 451.264,A -85,B 0,C 180,E1 -26029.522,E2 -26029.522} C_VEL
LIN {X 0,Y 118.674,Z 446.026,A -85,B 0,C 180,E1 -26034.493,E2 -26034.493} C_VEL
LIN {X 0,Y 122.489,Z 439.128,A -85,B 0,C 180,E1 -26039.191,E2 -26039.191} C_VEL
LIN {X 0,Y 126.403,Z 431.617,A -85,B 0,C 180,E1 -26042.828,E2 -26042.828} C_VEL
LIN {X 0,Y 129.371,Z 425.254,A -85,B 0,C 180,E1 -26045.247,E2 -26045.247} C_VEL
LIN {X 0,Y 132.585,Z 417.515,A -85,B 0,C 180,E1 -26047.561,E2 -26047.561} C_VEL
LIN {X 0,Y 135.532,Z 409.405,A -85,B 0,C 180,E1 -26049.438,E2 -26049.438} C_VEL
LIN {X 0,Y 138.114,Z 400.993,A -85,B 0,C 180,E1 -26050.933,E2 -26050.933} C_VEL
LIN {X 0,Y 140.751,Z 390.755,A -85,B 0,C 180,E1 -26052.229,E2 -26052.229} C_VEL
LIN {X 0,Y 142.753,Z 377.869,A -85,B 0,C 180,E1 -26053.349,E2 -26053.349} C_VEL
LIN {X 0,Y 143.718,Z 365.727,A -85,B 0,C 180,E1 -26053.965,E2 -26053.965} C_VEL
LIN {X 0,Y 143.42,Z 360.197,A -85,B 0,C 180,E1 -26054.454,E2 -26054.454} C_VEL
LIN {X 0,Y 142.814,Z 356.518,A -85,B 0,C 180,E1 -26054.943,E2 -26054.943} C_VEL
LIN {X 0,Y 141.009,Z 351.55,A -85,B 0,C 180,E1 -26056.023,E2 -26056.023} C_VEL
LIN {X 0,Y 138.588,Z 347.192,A -85,B 0,C 180,E1 -26057.378,E2 -26057.378} C_VEL
LIN {X 0,Y 131.659,Z 336.057,A -85,B 0,C 180,E1 -26061.654,E2 -26061.654} C_VEL
LIN {X 0,Y 128.004,Z 328.578,A -85,B 0,C 180,E1 -26064.434,E2 -26064.434} C_VEL
LIN {X 0,Y 123.709,Z 322.226,A -85,B 0,C 180,E1 -26067.939,E2 -26067.939} C_VEL
LIN {X 0,Y 120.7,Z 318.081,A -85,B 0,C 180,E1 -26070.743,E2 -26070.743} C_VEL
LIN {X 0,Y 118.237,Z 315.167,A -85,B 0,C 180,E1 -26073.288,E2 -26073.288} C_VEL
LIN {X 0,Y 116.991,Z 313.196,A -85,B 0,C 180,E1 -26074.777,E2 -26074.777} C_VEL
LIN {X 0,Y 114.633,Z 311.102,A -85,B 0,C 180,E1 -26077.686,E2 -26077.686} C_VEL
LIN {X 0,Y 113.048,Z 307.984,A -85,B 0,C 180,E1 -26080.243,E2 -26080.243} C_VEL
LIN {X 0,Y 109.847,Z 305.752,A -85,B 0,C 180,E1 -26085.999,E2 -26085.999} C_VEL
LIN {X 0,Y 108.332,Z 302.362,A -85,B 0,C 180,E1 -26090.784,E2 -26090.784} C_VEL
LIN {X 0,Y 108.24,Z 301.766,A -85,B 0,C 180,E1 -26091.6,E2 -26091.6} C_VEL
LIN {X 0,Y 108.879,Z 301.714,A -85,B 0,C 180,E1 -26100,E2 -26100} C_VEL
LIN {X 0,Y 108.274,Z 301.956,A -85,B 0,C 180,E1 -26109.693,E2 -26109.693} C_VEL
LIN {X 0,Y 109.233,Z 304.862,A -85,B 0,C 180,E1 -26113.255,E2 -26113.255} C_VEL
LIN {X 0,Y 111.384,Z 307.086,A -85,B 0,C 180,E1 -26117.915,E2 -26117.915} C_VEL
LIN {X 0,Y 113.056,Z 307.967,A -85,B 0,C 180,E1 -26120.587,E2 -26120.587} C_VEL
LIN {X 0,Y 114.456,Z 310.937,A -85,B 0,C 180,E1 -26122.898,E2 -26122.898} C_VEL
LIN {X 0,Y 116.822,Z 313.11,A -85,B 0,C 180,E1 -26125.86,E2 -26125.86} C_VEL
LIN {X 0,Y 117.427,Z 313.692,A -85,B 0,C 180,E1 -26126.552,E2 -26126.552} C_VEL
LIN {X 0,Y 119.59,Z 317.015,A -85,B 0,C 180,E1 -26129.002,E2 -26129.002} C_VEL
LIN {X 0,Y 121.235,Z 318.774,A -85,B 0,C 180,E1 -26130.601,E2 -26130.601} C_VEL
LIN {X 0,Y 124.889,Z 324.01,A -85,B 0,C 180,E1 -26133.907,E2 -26133.907} C_VEL
LIN {X 0,Y 127.744,Z 328.263,A -85,B 0,C 180,E1 -26136.198,E2 -26136.198} C_VEL
LIN {X 0,Y 132.366,Z 335.601,A -85,B 0,C 180,E1 -26139.509,E2 -26139.509} C_VEL
LIN {X 0,Y 137.159,Z 344.369,A -85,B 0,C 180,E1 -26142.586,E2 -26142.586} C_VEL
LIN {X 0,Y 139.729,Z 349.792,A -85,B 0,C 180,E1 -26144.133,E2 -26144.133} C_VEL
LIN {X 0,Y 138.477,Z 366.762,A -85,B 0,C 180,E1 -26145.007,E2 -26145.007} C_VEL
LIN {X 0,Y 136.655,Z 379.188,A -85,B 0,C 180,E1 -26146.161,E2 -26146.161} C_VEL
LIN {X 0,Y 134.897,Z 387.71,A -85,B 0,C 180,E1 -26147.366,E2 -26147.366} C_VEL
LIN {X 0,Y 132.394,Z 396.477,A -85,B 0,C 180,E1 -26148.933,E2 -26148.933} C_VEL
LIN {X 0,Y 129.377,Z 404.831,A -85,B 0,C 180,E1 -26150.838,E2 -26150.838} C_VEL
LIN {X 0,Y 126.119,Z 412.712,A -85,B 0,C 180,E1 -26153.197,E2 -26153.197} C_VEL
LIN {X 0,Y 122.75,Z 420.051,A -85,B 0,C 180,E1 -26156.065,E2 -26156.065} C_VEL
LIN {X 0,Y 118.735,Z 427.494,A -85,B 0,C 180,E1 -26159.791,E2 -26159.791} C_VEL
LIN {X 0,Y 114.554,Z 434.307,A -85,B 0,C 180,E1 -26164.565,E2 -26164.565} C_VEL
LIN {X 0,Y 111.183,Z 439.452,A -85,B 0,C 180,E1 -26169.654,E2 -26169.654} C_VEL
LIN {X 0,Y 109.397,Z 442.086,A -85,B 0,C 180,E1 -26173.194,E2 -26173.194} C_VEL
LIN {X 0,Y 107.21,Z 445.327,A -85,B 0,C 180,E1 -26179.518,E2 -26179.518} C_VEL
LIN {X 0,Y 105.941,Z 447.015,A -85,B 0,C 180,E1 -26186.194,E2 -26186.194} C_VEL
LIN {X 0,Y 105.755,Z 447.316,A -85,B 0,C 180,E1 -26189.998,E2 -26189.998} C_VEL
LIN {X 0,Y 105.937,Z 447.035,A -85,B 0,C 180,E1 -26193.802,E2 -26193.802} C_VEL
LIN {X 0,Y 107.007,Z 445.671,A -85,B 0,C 180,E1 -26199.879,E2 -26199.879} C_VEL
LIN {X 0,Y 108.676,Z 443.367,A -85,B 0,C 180,E1 -26204.989,E2 -26204.989} C_VEL
LIN {X 0,Y 111.161,Z 439.641,A -85,B 0,C 180,E1 -26210.346,E2 -26210.346} C_VEL
LIN {X 0,Y 114.497,Z 434.549,A -85,B 0,C 180,E1 -26215.445,E2 -26215.445} C_VEL
LIN {X 0,Y 117.899,Z 429.063,A -85,B 0,C 180,E1 -26219.456,E2 -26219.456} C_VEL
LIN {X 0,Y 121.854,Z 422.153,A -85,B 0,C 180,E1 -26223.222,E2 -26223.222} C_VEL
LIN {X 0,Y 125.582,Z 414.23,A -85,B 0,C 180,E1 -26226.483,E2 -26226.483} C_VEL
LIN {X 0,Y 128.872,Z 406.659,A -85,B 0,C 180,E1 -26228.838,E2 -26228.838} C_VEL
LIN {X 0,Y 131.855,Z 398.714,A -85,B 0,C 180,E1 -26230.761,E2 -26230.761} C_VEL
LIN {X 0,Y 134.318,Z 390.502,A -85,B 0,C 180,E1 -26232.348,E2 -26232.348} C_VEL
LIN {X 0,Y 136.231,Z 382.638,A -85,B 0,C 180,E1 -26233.526,E2 -26233.526} C_VEL
LIN {X 0,Y 137.827,Z 373.318,A -85,B 0,C 180,E1 -26234.611,E2 -26234.611} C_VEL
LIN {X 0,Y 138.955,Z 363.819,A -85,B 0,C 180,E1 -26235.338,E2 -26235.338} C_VEL
LIN {X 0,Y 139.967,Z 350.128,A -85,B 0,C 180,E1 -26235.993,E2 -26235.993} C_VEL
LIN {X 0,Y 135.397,Z 340.885,A -85,B 0,C 180,E1 -26238.79,E2 -26238.79} C_VEL
LIN {X 0,Y 130.88,Z 333.014,A -85,B 0,C 180,E1 -26241.818,E2 -26241.818} C_VEL
LIN {X 0,Y 126.304,Z 325.953,A -85,B 0,C 180,E1 -26245.269,E2 -26245.269} C_VEL
LIN {X 0,Y 123.51,Z 321.948,A -85,B 0,C 180,E1 -26247.642,E2 -26247.642} C_VEL
LIN {X 0,Y 120.735,Z 318.05,A -85,B 0,C 180,E1 -26250.276,E2 -26250.276} C_VEL
LIN {X 0,Y 118.252,Z 315.148,A -85,B 0,C 180,E1 -26252.873,E2 -26252.873} C_VEL
LIN {X 0,Y 117.224,Z 313.314,A -85,B 0,C 180,E1 -26254.141,E2 -26254.141} C_VEL
LIN {X 0,Y 114.651,Z 311.103,A -85,B 0,C 180,E1 -26257.342,E2 -26257.342} C_VEL
LIN {X 0,Y 113.046,Z 307.889,A -85,B 0,C 180,E1 -26260.005,E2 -26260.005} C_VEL
LIN {X 0,Y 110,Z 305.918,A -85,B 0,C 180,E1 -26265.605,E2 -26265.605} C_VEL
LIN {X 0,Y 108.337,Z 302.425,A -85,B 0,C 180,E1 -26271.137,E2 -26271.137} C_VEL
LIN {X 0,Y 108.262,Z 301.8,A -85,B 0,C 180,E1 -26272.071,E2 -26272.071} C_VEL
LIN {X 0,Y 108.892,Z 301.714,A -85,B 0,C 180,E1 -26280,E2 -26280} C_VEL
LIN {X 0,Y 108.302,Z 301.988,A -85,B 0,C 180,E1 -26287.808,E2 -26287.808} C_VEL
LIN {X 0,Y 108.827,Z 303.857,A -85,B 0,C 180,E1 -26290.229,E2 -26290.229} C_VEL
LIN {X 0,Y 110.903,Z 306.787,A -85,B 0,C 180,E1 -26295.624,E2 -26295.624} C_VEL
LIN {X 0,Y 113.112,Z 308.078,A -85,B 0,C 180,E1 -26299.391,E2 -26299.391} C_VEL
LIN {X 0,Y 114.517,Z 310.892,A -85,B 0,C 180,E1 -26301.728,E2 -26301.728} C_VEL
LIN {X 0,Y 116.777,Z 313.09,A -85,B 0,C 180,E1 -26304.632,E2 -26304.632} C_VEL
LIN {X 0,Y 117.552,Z 313.88,A -85,B 0,C 180,E1 -26305.538,E2 -26305.538} C_VEL
LIN {X 0,Y 120.054,Z 317.476,A -85,B 0,C 180,E1 -26308.339,E2 -26308.339} C_VEL
LIN {X 0,Y 121.417,Z 318.945,A -85,B 0,C 180,E1 -26309.663,E2 -26309.663} C_VEL
LIN {X 0,Y 124.859,Z 323.88,A -85,B 0,C 180,E1 -26312.804,E2 -26312.804} C_VEL
LIN {X 0,Y 128.004,Z 328.493,A -85,B 0,C 180,E1 -26315.336,E2 -26315.336} C_VEL
LIN {X 0,Y 130.677,Z 333.798,A -85,B 0,C 180,E1 -26317.405,E2 -26317.405} C_VEL
LIN {X 0,Y 135.038,Z 343.83,A -85,B 0,C 180,E1 -26320.537,E2 -26320.537} C_VEL
LIN {X 0,Y 138.112,Z 352.553,A -85,B 0,C 180,E1 -26322.643,E2 -26322.643} C_VEL
LIN {X 0,Y 138.815,Z 367.045,A -85,B 0,C 180,E1 -26324.014,E2 -26324.014} C_VEL
LIN {X 0,Y 137.369,Z 381.289,A -85,B 0,C 180,E1 -26324.81,E2 -26324.81} C_VEL
LIN {X 0,Y 135.491,Z 391.294,A -85,B 0,C 180,E1 -26325.76,E2 -26325.76} C_VEL
LIN {X 0,Y 133.453,Z 399.316,A -85,B 0,C 180,E1 -26326.797,E2 -26326.797} C_VEL
LIN {X 0,Y 130.678,Z 407.98,A -85,B 0,C 180,E1 -26328.279,E2 -26328.279} C_VEL
LIN {X 0,Y 127.566,Z 416.273,A -85,B 0,C 180,E1 -26330.177,E2 -26330.177} C_VEL
LIN {X 0,Y 124.276,Z 423.693,A -85,B 0,C 180,E1 -26332.346,E2 -26332.346} C_VEL
LIN {X 0,Y 121.353,Z 429.774,A -85,B 0,C 180,E1 -26334.612,E2 -26334.612} C_VEL
LIN {X 0,Y 117.936,Z 436.111,A -85,B 0,C 180,E1 -26337.569,E2 -26337.569} C_VEL
LIN {X 0,Y 114.902,Z 441.383,A -85,B 0,C 180,E1 -26340.706,E2 -26340.706} C_VEL
LIN {X 0,Y 112.232,Z 445.784,A -85,B 0,C 180,E1 -26344.004,E2 -26344.004} C_VEL
LIN {X 0,Y 108.983,Z 450.987,A -85,B 0,C 180,E1 -26349.228,E2 -26349.228} C_VEL
LIN {X 0,Y 106.839,Z 454.827,A -85,B 0,C 180,E1 -26354.746,E2 -26354.746} C_VEL
LIN {X 0,Y 105.916,Z 456.597,A -85,B 0,C 180,E1 -26358.52,E2 -26358.52} C_VEL
LIN {X 0,Y 105.451,Z 457.872,A -85,B 0,C 180,E1 -26362.342,E2 -26362.342} C_VEL
LIN {X 0,Y 105.444,Z 458.904,A -85,B 0,C 180,E1 -26368.76,E2 -26368.76} C_VEL
LIN {X 0,Y 105.444,Z 458.892,A -85,B 0,C 180,E1 -26371.244,E2 -26371.244} C_VEL
LIN {X 0,Y 105.452,Z 457.834,A -85,B 0,C 180,E1 -26377.662,E2 -26377.662} C_VEL
LIN {X 0,Y 105.917,Z 456.533,A -85,B 0,C 180,E1 -26381.484,E2 -26381.484} C_VEL
LIN {X 0,Y 107.455,Z 453.565,A -85,B 0,C 180,E1 -26387.119,E2 -26387.119} C_VEL
LIN {X 0,Y 108.983,Z 450.868,A -85,B 0,C 180,E1 -26390.776,E2 -26390.776} C_VEL
LIN {X 0,Y 112.23,Z 445.631,A -85,B 0,C 180,E1 -26396.001,E2 -26396.001} C_VEL
LIN {X 0,Y 116.323,Z 438.733,A -85,B 0,C 180,E1 -26400.903,E2 -26400.903} C_VEL
LIN {X 0,Y 120.49,Z 431.222,A -85,B 0,C 180,E1 -26404.662,E2 -26404.662} C_VEL
LIN {X 0,Y 124.168,Z 423.661,A -85,B 0,C 180,E1 -26407.556,E2 -26407.556} C_VEL
LIN {X 0,Y 127.51,Z 415.883,A -85,B 0,C 180,E1 -26409.849,E2 -26409.849} C_VEL
LIN {X 0,Y 131.19,Z 406,A -85,B 0,C 180,E1 -26412.041,E2 -26412.041} C_VEL
LIN {X 0,Y 134.213,Z 395.932,A -85,B 0,C 180,E1 -26413.61,E2 -26413.61} C_VEL
LIN {X 0,Y 136.581,Z 385.045,A -85,B 0,C 180,E1 -26414.773,E2 -26414.773} C_VEL
LIN {X 0,Y 137.798,Z 376.267,A -85,B 0,C 180,E1 -26415.446,E2 -26415.446} C_VEL
LIN {X 0,Y 138.61,Z 366.055,A -85,B 0,C 180,E1 -26415.983,E2 -26415.983} C_VEL
LIN {X 0,Y 137.8,Z 351.759,A -85,B 0,C 180,E1 -26417.387,E2 -26417.387} C_VEL
LIN {X 0,Y 134.119,Z 341.803,A -85,B 0,C 180,E1 -26419.897,E2 -26419.897} C_VEL
LIN {X 0,Y 131.659,Z 336.057,A -85,B 0,C 180,E1 -26421.654,E2 -26421.654} C_VEL
LIN {X 0,Y 129.976,Z 333.672,A -85,B 0,C 180,E1 -26422.799,E2 -26422.799} C_VEL
LIN {X 0,Y 127.938,Z 332.108,A -85,B 0,C 180,E1 -26424.146,E2 -26424.146} C_VEL
LIN {X 0,Y 121.681,Z 328.779,A -85,B 0,C 180,E1 -26428.743,E2 -26428.743} C_VEL
LIN {X 0,Y 121.093,Z 328.213,A -85,B 0,C 180,E1 -26429.26,E2 -26429.26} C_VEL
LIN {X 0,Y 118.271,Z 324.223,A -85,B 0,C 180,E1 -26432.099,E2 -26432.099} C_VEL
LIN {X 0,Y 115.743,Z 320.853,A -85,B 0,C 180,E1 -26434.99,E2 -26434.99} C_VEL
LIN {X 0,Y 114.883,Z 319.664,A -85,B 0,C 180,E1 -26436.084,E2 -26436.084} C_VEL
LIN {X 0,Y 112.402,Z 316.919,A -85,B 0,C 180,E1 -26439.53,E2 -26439.53} C_VEL
LIN {X 0,Y 111.258,Z 314.562,A -85,B 0,C 180,E1 -26441.589,E2 -26441.589} C_VEL
LIN {X 0,Y 108.653,Z 312.632,A -85,B 0,C 180,E1 -26446.675,E2 -26446.675} C_VEL
LIN {X 0,Y 107.188,Z 309.199,A -85,B 0,C 180,E1 -26451.754,E2 -26451.754} C_VEL
LIN {X 0,Y 107.052,Z 308.753,A -85,B 0,C 180,E1 -26452.456,E2 -26452.456} C_VEL
LIN {X 0,Y 106.087,Z 308.249,A -85,B 0,C 180,E1 -26460,E2 -26460} C_VEL
LIN {X 0,Y 107.156,Z 308.951,A -85,B 0,C 180,E1 -26468.843,E2 -26468.843} C_VEL
LIN {X 0,Y 108.063,Z 311.729,A -85,B 0,C 180,E1 -26472.524,E2 -26472.524} C_VEL
LIN {X 0,Y 110.065,Z 313.935,A -85,B 0,C 180,E1 -26477.177,E2 -26477.177} C_VEL
LIN {X 0,Y 111.382,Z 314.804,A -85,B 0,C 180,E1 -26479.466,E2 -26479.466} C_VEL
LIN {X 0,Y 113.132,Z 318.006,A -85,B 0,C 180,E1 -26482.422,E2 -26482.422} C_VEL
LIN {X 0,Y 115.384,Z 320.188,A -85,B 0,C 180,E1 -26485.358,E2 -26485.358} C_VEL
LIN {X 0,Y 117.824,Z 323.765,A -85,B 0,C 180,E1 -26488.259,E2 -26488.259} C_VEL
LIN {X 0,Y 119.021,Z 325.302,A -85,B 0,C 180,E1 -26489.518,E2 -26489.518} C_VEL
LIN {X 0,Y 122.171,Z 329.928,A -85,B 0,C 180,E1 -26492.574,E2 -26492.574} C_VEL
LIN {X 0,Y 126.317,Z 336.376,A -85,B 0,C 180,E1 -26496.072,E2 -26496.072} C_VEL
LIN {X 0,Y 131.093,Z 344.827,A -85,B 0,C 180,E1 -26499.609,E2 -26499.609} C_VEL
LIN {X 0,Y 134.733,Z 352.355,A -85,B 0,C 180,E1 -26502.066,E2 -26502.066} C_VEL
LIN {X 0,Y 133.457,Z 368.131,A -85,B 0,C 180,E1 -26502.912,E2 -26502.912} C_VEL
LIN {X 0,Y 131.639,Z 379.587,A -85,B 0,C 180,E1 -26504.025,E2 -26504.025} C_VEL
LIN {X 0,Y 129.777,Z 388.107,A -85,B 0,C 180,E1 -26505.248,E2 -26505.248} C_VEL
LIN {X 0,Y 127.155,Z 396.872,A -85,B 0,C 180,E1 -26506.842,E2 -26506.842} C_VEL
LIN {X 0,Y 123.974,Z 405.225,A -85,B 0,C 180,E1 -26508.773,E2 -26508.773} C_VEL
LIN {X 0,Y 120.536,Z 413.105,A -85,B 0,C 180,E1 -26511.184,E2 -26511.184} C_VEL
LIN {X 0,Y 116.955,Z 420.444,A -85,B 0,C 180,E1 -26514.132,E2 -26514.132} C_VEL
LIN {X 0,Y 112.685,Z 427.886,A -85,B 0,C 180,E1 -26517.984,E2 -26517.984} C_VEL
LIN {X 0,Y 108.194,Z 434.7,A -85,B 0,C 180,E1 -26522.952,E2 -26522.952} C_VEL
LIN {X 0,Y 104.564,Z 439.845,A -85,B 0,C 180,E1 -26528.303,E2 -26528.303} C_VEL
LIN {X 0,Y 102.631,Z 442.479,A -85,B 0,C 180,E1 -26532.05,E2 -26532.05} C_VEL
LIN {X 0,Y 100.542,Z 445.356,A -85,B 0,C 180,E1 -26537.893,E2 -26537.893} C_VEL
LIN {X 0,Y 99.48,Z 446.616,A -85,B 0,C 180,E1 -26541.875,E2 -26541.875} C_VEL
LIN {X 0,Y 98.88,Z 447.406,A -85,B 0,C 180,E1 -26545.922,E2 -26545.922} C_VEL
LIN {X 0,Y 98.67,Z 447.707,A -85,B 0,C 180,E1 -26549.998,E2 -26549.998} C_VEL
LIN {X 0,Y 98.879,Z 447.425,A -85,B 0,C 180,E1 -26554.074,E2 -26554.074} C_VEL
LIN {X 0,Y 99.887,Z 446.247,A -85,B 0,C 180,E1 -26559.924,E2 -26559.924} C_VEL
LIN {X 0,Y 101.852,Z 443.757,A -85,B 0,C 180,E1 -26566.02,E2 -26566.02} C_VEL
LIN {X 0,Y 104.547,Z 440.031,A -85,B 0,C 180,E1 -26571.697,E2 -26571.697} C_VEL
LIN {X 0,Y 108.142,Z 434.939,A -85,B 0,C 180,E1 -26577.058,E2 -26577.058} C_VEL
LIN {X 0,Y 111.801,Z 429.451,A -85,B 0,C 180,E1 -26581.237,E2 -26581.237} C_VEL
LIN {X 0,Y 116.008,Z 422.54,A -85,B 0,C 180,E1 -26585.134,E2 -26585.134} C_VEL
LIN {X 0,Y 119.97,Z 414.617,A -85,B 0,C 180,E1 -26588.491,E2 -26588.491} C_VEL
LIN {X 0,Y 123.44,Z 407.046,A -85,B 0,C 180,E1 -26590.898,E2 -26590.898} C_VEL
LIN {X 0,Y 126.586,Z 399.099,A -85,B 0,C 180,E1 -26592.85,E2 -26592.85} C_VEL
LIN {X 0,Y 129.17,Z 390.887,A -85,B 0,C 180,E1 -26594.466,E2 -26594.466} C_VEL
LIN {X 0,Y 131.366,Z 382.267,A -85,B 0,C 180,E1 -26595.748,E2 -26595.748} C_VEL
LIN {X 0,Y 132.998,Z 373.044,A -85,B 0,C 180,E1 -26596.811,E2 -26596.811} C_VEL
LIN {X 0,Y 134.106,Z 363.943,A -85,B 0,C 180,E1 -26597.501,E2 -26597.501} C_VEL
LIN {X 0,Y 134.982,Z 352.648,A -85,B 0,C 180,E1 -26598.061,E2 -26598.061} C_VEL
LIN {X 0,Y 130.537,Z 343.656,A -85,B 0,C 180,E1 -26601.082,E2 -26601.082} C_VEL
LIN {X 0,Y 125.653,Z 335.126,A -85,B 0,C 180,E1 -26604.796,E2 -26604.796} C_VEL
LIN {X 0,Y 121.063,Z 328.12,A -85,B 0,C 180,E1 -26608.838,E2 -26608.838} C_VEL
LIN {X 0,Y 118.325,Z 324.238,A -85,B 0,C 180,E1 -26611.629,E2 -26611.629} C_VEL
LIN {X 0,Y 115.758,Z 320.809,A -85,B 0,C 180,E1 -26614.609,E2 -26614.609} C_VEL
LIN {X 0,Y 115.124,Z 319.772,A -85,B 0,C 180,E1 -26615.447,E2 -26615.447} C_VEL
LIN {X 0,Y 112.654,Z 317.238,A -85,B 0,C 180,E1 -26618.858,E2 -26618.858} C_VEL
LIN {X 0,Y 111.391,Z 314.677,A -85,B 0,C 180,E1 -26621.148,E2 -26621.148} C_VEL
LIN {X 0,Y 108.566,Z 312.458,A -85,B 0,C 180,E1 -26626.949,E2 -26626.949} C_VEL
LIN {X 0,Y 107.098,Z 308.79,A -85,B 0,C 180,E1 -26632.932,E2 -26632.932} C_VEL
LIN {X 0,Y 106.419,Z 308.376,A -85,B 0,C 180,E1 -26640,E2 -26640} C_VEL
LIN {X 0,Y 107.188,Z 308.966,A -85,B 0,C 180,E1 -26646.825,E2 -26646.825} C_VEL
LIN {X 0,Y 108.83,Z 312.797,A -85,B 0,C 180,E1 -26653.019,E2 -26653.019} C_VEL
LIN {X 0,Y 111.455,Z 314.883,A -85,B 0,C 180,E1 -26658.259,E2 -26658.259} C_VEL
LIN {X 0,Y 113.425,Z 318.273,A -85,B 0,C 180,E1 -26661.586,E2 -26661.586} C_VEL
LIN {X 0,Y 115.585,Z 320.463,A -85,B 0,C 180,E1 -26664.425,E2 -26664.425} C_VEL
LIN {X 0,Y 118.145,Z 324.064,A -85,B 0,C 180,E1 -26667.452,E2 -26667.452} C_VEL
LIN {X 0,Y 119.239,Z 325.535,A -85,B 0,C 180,E1 -26668.613,E2 -26668.613} C_VEL
LIN {X 0,Y 122.323,Z 330.07,A -85,B 0,C 180,E1 -26671.619,E2 -26671.619} C_VEL
LIN {X 0,Y 125.126,Z 334.382,A -85,B 0,C 180,E1 -26674.05,E2 -26674.05} C_VEL
LIN {X 0,Y 128.663,Z 342.305,A -85,B 0,C 180,E1 -26677.005,E2 -26677.005} C_VEL
LIN {X 0,Y 132.018,Z 350.905,A -85,B 0,C 180,E1 -26679.591,E2 -26679.591} C_VEL
LIN {X 0,Y 133.43,Z 355.498,A -85,B 0,C 180,E1 -26680.68,E2 -26680.68} C_VEL
LIN {X 0,Y 133.844,Z 368.404,A -85,B 0,C 180,E1 -26681.901,E2 -26681.901} C_VEL
LIN {X 0,Y 132.327,Z 381.647,A -85,B 0,C 180,E1 -26682.692,E2 -26682.692} C_VEL
LIN {X 0,Y 130.361,Z 391.487,A -85,B 0,C 180,E1 -26683.655,E2 -26683.655} C_VEL
LIN {X 0,Y 128.371,Z 398.93,A -85,B 0,C 180,E1 -26684.628,E2 -26684.628} C_VEL
LIN {X 0,Y 125.477,Z 407.593,A -85,B 0,C 180,E1 -26686.124,E2 -26686.124} C_VEL
LIN {X 0,Y 122.185,Z 415.884,A -85,B 0,C 180,E1 -26688.039,E2 -26688.039} C_VEL
LIN {X 0,Y 118.77,Z 423.226,A -85,B 0,C 180,E1 -26690.225,E2 -26690.225} C_VEL
LIN {X 0,Y 115.615,Z 429.383,A -85,B 0,C 180,E1 -26692.566,E2 -26692.566} C_VEL
LIN {X 0,Y 112.016,Z 435.722,A -85,B 0,C 180,E1 -26695.623,E2 -26695.623} C_VEL
LIN {X 0,Y 108.729,Z 440.99,A -85,B 0,C 180,E1 -26698.864,E2 -26698.864} C_VEL
LIN {X 0,Y 105.883,Z 445.392,A -85,B 0,C 180,E1 -26702.316,E2 -26702.316} C_VEL
LIN {X 0,Y 102.351,Z 450.595,A -85,B 0,C 180,E1 -26707.814,E2 -26707.814} C_VEL
LIN {X 0,Y 99.983,Z 454.435,A -85,B 0,C 180,E1 -26713.672,E2 -26713.672} C_VEL
LIN {X 0,Y 98.949,Z 456.204,A -85,B 0,C 180,E1 -26717.699,E2 -26717.699} C_VEL
LIN {X 0,Y 98.388,Z 457.479,A -85,B 0,C 180,E1 -26721.789,E2 -26721.789} C_VEL
LIN {X 0,Y 98.236,Z 458.277,A -85,B 0,C 180,E1 -26725.9,E2 -26725.9} C_VEL
LIN {X 0,Y 98.398,Z 458.555,A -85,B 0,C 180,E1 -26730.669,E2 -26730.669} C_VEL
LIN {X 0,Y 98.242,Z 458.265,A -85,B 0,C 180,E1 -26734.104,E2 -26734.104} C_VEL
LIN {X 0,Y 98.389,Z 457.44,A -85,B 0,C 180,E1 -26738.216,E2 -26738.216} C_VEL
LIN {X 0,Y 98.949,Z 456.139,A -85,B 0,C 180,E1 -26742.305,E2 -26742.305} C_VEL
LIN {X 0,Y 100.657,Z 453.17,A -85,B 0,C 180,E1 -26748.314,E2 -26748.314} C_VEL
LIN {X 0,Y 102.352,Z 450.474,A -85,B 0,C 180,E1 -26752.191,E2 -26752.191} C_VEL
LIN {X 0,Y 105.88,Z 445.237,A -85,B 0,C 180,E1 -26757.689,E2 -26757.689} C_VEL
LIN {X 0,Y 110.282,Z 438.338,A -85,B 0,C 180,E1 -26762.8,E2 -26762.8} C_VEL
LIN {X 0,Y 114.712,Z 430.827,A -85,B 0,C 180,E1 -26766.682,E2 -26766.682} C_VEL
LIN {X 0,Y 118.275,Z 423.935,A -85,B 0,C 180,E1 -26769.424,E2 -26769.424} C_VEL
LIN {X 0,Y 121.616,Z 416.722,A -85,B 0,C 180,E1 -26771.651,E2 -26771.651} C_VEL
LIN {X 0,Y 124.881,Z 408.611,A -85,B 0,C 180,E1 -26773.585,E2 -26773.585} C_VEL
LIN {X 0,Y 127.724,Z 400.197,A -85,B 0,C 180,E1 -26775.111,E2 -26775.111} C_VEL
LIN {X 0,Y 130.283,Z 391.146,A -85,B 0,C 180,E1 -26776.285,E2 -26776.285} C_VEL
LIN {X 0,Y 132.459,Z 379.838,A -85,B 0,C 180,E1 -26777.371,E2 -26777.371} C_VEL
LIN {X 0,Y 133.687,Z 366.631,A -85,B 0,C 180,E1 -26778.134,E2 -26778.134} C_VEL
LIN {X 0,Y 133.025,Z 354.295,A -85,B 0,C 180,E1 -26779.434,E2 -26779.434} C_VEL
LIN {X 0,Y 129.561,Z 344.613,A -85,B 0,C 180,E1 -26782.07,E2 -26782.07} C_VEL
LIN {X 0,Y 125.151,Z 334.512,A -85,B 0,C 180,E1 -26785.684,E2 -26785.684} C_VEL
LIN {X 0,Y 121.093,Z 328.213,A -85,B 0,C 180,E1 -26789.26,E2 -26789.26} C_VEL
LIN {X 0,Y 117.772,Z 325.359,A -85,B 0,C 180,E1 -26792.408,E2 -26792.408} C_VEL
LIN {X 0,Y 113.061,Z 322.872,A -85,B 0,C 180,E1 -26797.692,E2 -26797.692} C_VEL
LIN {X 0,Y 109.243,Z 321.106,A -85,B 0,C 180,E1 -26803.475,E2 -26803.475} C_VEL
LIN {X 0,Y 107.035,Z 318.832,A -85,B 0,C 180,E1 -26808.64,E2 -26808.64} C_VEL
LIN {X 0,Y 105.969,Z 315.753,A -85,B 0,C 180,E1 -26813.336,E2 -26813.336} C_VEL
LIN {X 0,Y 105.223,Z 315.286,A -85,B 0,C 180,E1 -26820,E2 -26820} C_VEL
LIN {X 0,Y 106.059,Z 315.965,A -85,B 0,C 180,E1 -26827.975,E2 -26827.975} C_VEL
LIN {X 0,Y 107.272,Z 319.253,A -85,B 0,C 180,E1 -26832.901,E2 -26832.901} C_VEL
LIN {X 0,Y 109.818,Z 321.659,A -85,B 0,C 180,E1 -26838.421,E2 -26838.421} C_VEL
LIN {X 0,Y 111.821,Z 325.036,A -85,B 0,C 180,E1 -26841.935,E2 -26841.935} C_VEL
LIN {X 0,Y 113.428,Z 326.733,A -85,B 0,C 180,E1 -26844.17,E2 -26844.17} C_VEL
LIN {X 0,Y 116.147,Z 330.573,A -85,B 0,C 180,E1 -26847.568,E2 -26847.568} C_VEL
LIN {X 0,Y 120.127,Z 336.816,A -85,B 0,C 180,E1 -26851.773,E2 -26851.773} C_VEL
LIN {X 0,Y 124.609,Z 344.294,A -85,B 0,C 180,E1 -26855.743,E2 -26855.743} C_VEL
LIN {X 0,Y 129.262,Z 353.426,A -85,B 0,C 180,E1 -26859.354,E2 -26859.354} C_VEL
LIN {X 0,Y 129.876,Z 354.856,A -85,B 0,C 180,E1 -26859.81,E2 -26859.81} C_VEL
LIN {X 0,Y 128.529,Z 370.331,A -85,B 0,C 180,E1 -26860.75,E2 -26860.75} C_VEL
LIN {X 0,Y 126.597,Z 381.026,A -85,B 0,C 180,E1 -26861.869,E2 -26861.869} C_VEL
LIN {X 0,Y 124.317,Z 390.367,A -85,B 0,C 180,E1 -26863.291,E2 -26863.291} C_VEL
LIN {X 0,Y 121.521,Z 398.763,A -85,B 0,C 180,E1 -26864.888,E2 -26864.888} C_VEL
LIN {X 0,Y 118.211,Z 406.844,A -85,B 0,C 180,E1 -26866.864,E2 -26866.864} C_VEL
LIN {X 0,Y 114.575,Z 414.517,A -85,B 0,C 180,E1 -26869.325,E2 -26869.325} C_VEL
LIN {X 0,Y 110.33,Z 422.531,A -85,B 0,C 180,E1 -26872.759,E2 -26872.759} C_VEL
LIN {X 0,Y 105.883,Z 429.548,A -85,B 0,C 180,E1 -26876.796,E2 -26876.796} C_VEL
LIN {X 0,Y 101.939,Z 435.092,A -85,B 0,C 180,E1 -26881.142,E2 -26881.142} C_VEL
LIN {X 0,Y 98.023,Z 440.237,A -85,B 0,C 180,E1 -26886.773,E2 -26886.773} C_VEL
LIN {X 0,Y 95.928,Z 442.87,A -85,B 0,C 180,E1 -26890.748,E2 -26890.748} C_VEL
LIN {X 0,Y 93.622,Z 445.748,A -85,B 0,C 180,E1 -26896.983,E2 -26896.983} C_VEL
LIN {X 0,Y 92.48,Z 447.007,A -85,B 0,C 180,E1 -26901.255,E2 -26901.255} C_VEL
LIN {X 0,Y 91.812,Z 447.797,A -85,B 0,C 180,E1 -26905.608,E2 -26905.608} C_VEL
LIN {X 0,Y 91.582,Z 448.098,A -85,B 0,C 180,E1 -26909.998,E2 -26909.998} C_VEL
LIN {X 0,Y 91.811,Z 447.817,A -85,B 0,C 180,E1 -26914.388,E2 -26914.388} C_VEL
LIN {X 0,Y 92.692,Z 446.852,A -85,B 0,C 180,E1 -26919.709,E2 -26919.709} C_VEL
LIN {X 0,Y 95.051,Z 444.148,A -85,B 0,C 180,E1 -26927.2,E2 -26927.2} C_VEL
LIN {X 0,Y 97.988,Z 440.422,A -85,B 0,C 180,E1 -26933.231,E2 -26933.231} C_VEL
LIN {X 0,Y 101.892,Z 435.328,A -85,B 0,C 180,E1 -26938.868,E2 -26938.868} C_VEL
LIN {X 0,Y 105.805,Z 429.841,A -85,B 0,C 180,E1 -26943.227,E2 -26943.227} C_VEL
LIN {X 0,Y 110.284,Z 422.929,A -85,B 0,C 180,E1 -26947.255,E2 -26947.255} C_VEL
LIN {X 0,Y 114.524,Z 415.004,A -85,B 0,C 180,E1 -26950.692,E2 -26950.692} C_VEL
LIN {X 0,Y 118.183,Z 407.433,A -85,B 0,C 180,E1 -26953.144,E2 -26953.144} C_VEL
LIN {X 0,Y 121.5,Z 399.484,A -85,B 0,C 180,E1 -26955.117,E2 -26955.117} C_VEL
LIN {X 0,Y 124.216,Z 391.272,A -85,B 0,C 180,E1 -26956.754,E2 -26956.754} C_VEL
LIN {X 0,Y 126.621,Z 382.2,A -85,B 0,C 180,E1 -26958.109,E2 -26958.109} C_VEL
LIN {X 0,Y 128.446,Z 372.182,A -85,B 0,C 180,E1 -26959.244,E2 -26959.244} C_VEL
LIN {X 0,Y 129.874,Z 359.881,A -85,B 0,C 180,E1 -26960.051,E2 -26960.051} C_VEL
LIN {X 0,Y 130.157,Z 355.251,A -85,B 0,C 180,E1 -26960.293,E2 -26960.293} C_VEL
LIN {X 0,Y 125.523,Z 345.866,A -85,B 0,C 180,E1 -26963.84,E2 -26963.84} C_VEL
LIN {X 0,Y 121.056,Z 338.03,A -85,B 0,C 180,E1 -26967.737,E2 -26967.737} C_VEL
LIN {X 0,Y 117.429,Z 332.534,A -85,B 0,C 180,E1 -26971.393,E2 -26971.393} C_VEL
LIN {X 0,Y 115.798,Z 330.117,A -85,B 0,C 180,E1 -26973.264,E2 -26973.264} C_VEL
LIN {X 0,Y 113.142,Z 326.246,A -85,B 0,C 180,E1 -26976.732,E2 -26976.732} C_VEL
LIN {X 0,Y 110.684,Z 323.285,A -85,B 0,C 180,E1 -26980.527,E2 -26980.527} C_VEL
LIN {X 0,Y 109.747,Z 321.337,A -85,B 0,C 180,E1 -26982.411,E2 -26982.411} C_VEL
LIN {X 0,Y 107.406,Z 319.306,A -85,B 0,C 180,E1 -26987.675,E2 -26987.675} C_VEL
LIN {X 0,Y 106.138,Z 315.906,A -85,B 0,C 180,E1 -26993.312,E2 -26993.312} C_VEL
LIN {X 0,Y 105.553,Z 315.429,A -85,B 0,C 180,E1 -27000,E2 -27000} C_VEL
LIN {X 0,Y 106.136,Z 315.888,A -85,B 0,C 180,E1 -27005.938,E2 -27005.938} C_VEL
LIN {X 0,Y 107.856,Z 319.915,A -85,B 0,C 180,E1 -27012.849,E2 -27012.849} C_VEL
LIN {X 0,Y 109.908,Z 321.69,A -85,B 0,C 180,E1 -27017.202,E2 -27017.202} C_VEL
LIN {X 0,Y 112.138,Z 325.262,A -85,B 0,C 180,E1 -27021.122,E2 -27021.122} C_VEL
LIN {X 0,Y 113.614,Z 326.908,A -85,B 0,C 180,E1 -27023.196,E2 -27023.196} C_VEL
LIN {X 0,Y 116.337,Z 330.723,A -85,B 0,C 180,E1 -27026.617,E2 -27026.617} C_VEL
LIN {X 0,Y 119.992,Z 336.472,A -85,B 0,C 180,E1 -27030.528,E2 -27030.528} C_VEL
LIN {X 0,Y 122.329,Z 340.386,A -85,B 0,C 180,E1 -27032.726,E2 -27032.726} C_VEL
LIN {X 0,Y 126.389,Z 350.435,A -85,B 0,C 180,E1 -27036.397,E2 -27036.397} C_VEL
LIN {X 0,Y 128.866,Z 357.801,A -85,B 0,C 180,E1 -27038.492,E2 -27038.492} C_VEL
LIN {X 0,Y 129.119,Z 369.261,A -85,B 0,C 180,E1 -27039.613,E2 -27039.613} C_VEL
LIN {X 0,Y 127.62,Z 381.193,A -85,B 0,C 180,E1 -27040.336,E2 -27040.336} C_VEL
LIN {X 0,Y 125.79,Z 390.187,A -85,B 0,C 180,E1 -27041.198,E2 -27041.198} C_VEL
LIN {X 0,Y 123.493,Z 398.545,A -85,B 0,C 180,E1 -27042.286,E2 -27042.286} C_VEL
LIN {X 0,Y 120.449,Z 407.205,A -85,B 0,C 180,E1 -27043.778,E2 -27043.778} C_VEL
LIN {X 0,Y 117.015,Z 415.496,A -85,B 0,C 180,E1 -27045.719,E2 -27045.719} C_VEL
LIN {X 0,Y 113.155,Z 423.29,A -85,B 0,C 180,E1 -27048.08,E2 -27048.08} C_VEL
LIN {X 0,Y 109.065,Z 430.706,A -85,B 0,C 180,E1 -27051.08,E2 -27051.08} C_VEL
LIN {X 0,Y 104.387,Z 438.173,A -85,B 0,C 180,E1 -27055.094,E2 -27055.094} C_VEL
LIN {X 0,Y 100.393,Z 444.038,A -85,B 0,C 180,E1 -27059.503,E2 -27059.503} C_VEL
LIN {X 0,Y 96.948,Z 448.666,A -85,B 0,C 180,E1 -27064.22,E2 -27064.22} C_VEL
LIN {X 0,Y 94.772,Z 451.685,A -85,B 0,C 180,E1 -27068.238,E2 -27068.238} C_VEL
LIN {X 0,Y 93.152,Z 454.041,A -85,B 0,C 180,E1 -27072.437,E2 -27072.437} C_VEL
LIN {X 0,Y 92.016,Z 455.812,A -85,B 0,C 180,E1 -27076.756,E2 -27076.756} C_VEL
LIN {X 0,Y 91.349,Z 457.086,A -85,B 0,C 180,E1 -27081.151,E2 -27081.151} C_VEL
LIN {X 0,Y 91.157,Z 457.885,A -85,B 0,C 180,E1 -27085.581,E2 -27085.581} C_VEL
LIN {X 0,Y 91.363,Z 458.2,A -85,B 0,C 180,E1 -27090.002,E2 -27090.002} C_VEL
LIN {X 0,Y 91.16,Z 457.873,A -85,B 0,C 180,E1 -27094.424,E2 -27094.424} C_VEL
LIN {X 0,Y 91.349,Z 457.047,A -85,B 0,C 180,E1 -27098.854,E2 -27098.854} C_VEL
LIN {X 0,Y 92.016,Z 455.746,A -85,B 0,C 180,E1 -27103.248,E2 -27103.248} C_VEL
LIN {X 0,Y 93.914,Z 452.776,A -85,B 0,C 180,E1 -27109.682,E2 -27109.682} C_VEL
LIN {X 0,Y 95.799,Z 450.08,A -85,B 0,C 180,E1 -27113.799,E2 -27113.799} C_VEL
LIN {X 0,Y 99.641,Z 444.843,A -85,B 0,C 180,E1 -27119.588,E2 -27119.588} C_VEL
LIN {X 0,Y 104.382,Z 437.943,A -85,B 0,C 180,E1 -27124.913,E2 -27124.913} C_VEL
LIN {X 0,Y 109.077,Z 430.431,A -85,B 0,C 180,E1 -27128.92,E2 -27128.92} C_VEL
LIN {X 0,Y 112.375,Z 424.524,A -85,B 0,C 180,E1 -27131.368,E2 -27131.368} C_VEL
LIN {X 0,Y 116.411,Z 416.326,A -85,B 0,C 180,E1 -27133.972,E2 -27133.972} C_VEL
LIN {X 0,Y 119.839,Z 408.214,A -85,B 0,C 180,E1 -27135.925,E2 -27135.925} C_VEL
LIN {X 0,Y 122.816,Z 399.8,A -85,B 0,C 180,E1 -27137.458,E2 -27137.458} C_VEL
LIN {X 0,Y 125.329,Z 391.357,A -85,B 0,C 180,E1 -27138.555,E2 -27138.555} C_VEL
LIN {X 0,Y 127.362,Z 381.56,A -85,B 0,C 180,E1 -27139.537,E2 -27139.537} C_VEL
LIN {X 0,Y 128.834,Z 370.313,A -85,B 0,C 180,E1 -27140.25,E2 -27140.25} C_VEL
LIN {X 0,Y 128.931,Z 366.195,A -85,B 0,C 180,E1 -27140.551,E2 -27140.551} C_VEL
LIN {X 0,Y 128.54,Z 357.164,A -85,B 0,C 180,E1 -27141.541,E2 -27141.541} C_VEL
LIN {X 0,Y 125.578,Z 348.538,A -85,B 0,C 180,E1 -27144.057,E2 -27144.057} C_VEL
LIN {X 0,Y 121.863,Z 339.587,A -85,B 0,C 180,E1 -27147.44,E2 -27147.44} C_VEL
LIN {X 0,Y 117.964,Z 333.416,A -85,B 0,C 180,E1 -27151.232,E2 -27151.232} C_VEL
LIN {X 0,Y 115.789,Z 330.202,A -85,B 0,C 180,E1 -27153.651,E2 -27153.651} C_VEL
LIN {X 0,Y 113.072,Z 326.242,A -85,B 0,C 180,E1 -27157.141,E2 -27157.141} C_VEL
LIN {X 0,Y 110.606,Z 323.269,A -85,B 0,C 180,E1 -27160.877,E2 -27160.877} C_VEL
LIN {X 0,Y 109.644,Z 321.311,A -85,B 0,C 180,E1 -27162.756,E2 -27162.756} C_VEL
LIN {X 0,Y 109.243,Z 321.106,A -85,B 0,C 180,E1 -27163.475,E2 -27163.475} C_VEL
LIN {X 0,Y 107.273,Z 320.52,A -85,B 0,C 180,E1 -27167.539,E2 -27167.539} C_VEL
LIN {X 0,Y 105.157,Z 321.34,A -85,B 0,C 180,E1 -27173.891,E2 -27173.891} C_VEL
LIN {X 0,Y 104.35,Z 322.371,A -85,B 0,C 180,E1 -27180.441,E2 -27180.441} C_VEL
LIN {X 0,Y 105.001,Z 322.934,A -85,B 0,C 180,E1 -27187.123,E2 -27187.123} C_VEL
LIN {X 0,Y 106.278,Z 326.393,A -85,B 0,C 180,E1 -27192.665,E2 -27192.665} C_VEL
LIN {X 0,Y 108.33,Z 328.459,A -85,B 0,C 180,E1 -27197.4,E2 -27197.4} C_VEL
LIN {X 0,Y 110.399,Z 331.928,A -85,B 0,C 180,E1 -27201.251,E2 -27201.251} C_VEL
LIN {X 0,Y 111.637,Z 333.413,A -85,B 0,C 180,E1 -27203.105,E2 -27203.105} C_VEL
LIN {X 0,Y 114.598,Z 337.933,A -85,B 0,C 180,E1 -27207.043,E2 -27207.043} C_VEL
LIN {X 0,Y 118.255,Z 343.884,A -85,B 0,C 180,E1 -27211.085,E2 -27211.085} C_VEL
LIN {X 0,Y 122.783,Z 352.288,A -85,B 0,C 180,E1 -27215.331,E2 -27215.331} C_VEL
LIN {X 0,Y 125.271,Z 357.534,A -85,B 0,C 180,E1 -27217.421,E2 -27217.421} C_VEL
LIN {X 0,Y 123.872,Z 371.627,A -85,B 0,C 180,E1 -27218.357,E2 -27218.357} C_VEL
LIN {X 0,Y 121.981,Z 381.425,A -85,B 0,C 180,E1 -27219.389,E2 -27219.389} C_VEL
LIN {X 0,Y 119.578,Z 390.764,A -85,B 0,C 180,E1 -27220.823,E2 -27220.823} C_VEL
LIN {X 0,Y 116.633,Z 399.159,A -85,B 0,C 180,E1 -27222.423,E2 -27222.423} C_VEL
LIN {X 0,Y 113.156,Z 407.239,A -85,B 0,C 180,E1 -27224.416,E2 -27224.416} C_VEL
LIN {X 0,Y 109.307,Z 414.911,A -85,B 0,C 180,E1 -27226.908,E2 -27226.908} C_VEL
LIN {X 0,Y 104.78,Z 422.924,A -85,B 0,C 180,E1 -27230.414,E2 -27230.414} C_VEL
LIN {X 0,Y 100.049,Z 429.94,A -85,B 0,C 180,E1 -27234.58,E2 -27234.58} C_VEL
LIN {X 0,Y 95.805,Z 435.484,A -85,B 0,C 180,E1 -27239.1,E2 -27239.1} C_VEL
LIN {X 0,Y 91.546,Z 440.63,A -85,B 0,C 180,E1 -27245.022,E2 -27245.022} C_VEL
LIN {X 0,Y 89.261,Z 443.263,A -85,B 0,C 180,E1 -27249.246,E2 -27249.246} C_VEL
LIN {X 0,Y 86.736,Z 446.14,A -85,B 0,C 180,E1 -27255.929,E2 -27255.929} C_VEL
LIN {X 0,Y 85.501,Z 447.398,A -85,B 0,C 180,E1 -27260.535,E2 -27260.535} C_VEL
LIN {X 0,Y 84.758,Z 448.188,A -85,B 0,C 180,E1 -27265.241,E2 -27265.241} C_VEL
LIN {X 0,Y 84.514,Z 448.489,A -85,B 0,C 180,E1 -27269.998,E2 -27269.998} C_VEL
LIN {X 0,Y 84.757,Z 448.207,A -85,B 0,C 180,E1 -27274.754,E2 -27274.754} C_VEL
LIN {X 0,Y 85.499,Z 447.456,A -85,B 0,C 180,E1 -27279.46,E2 -27279.46} C_VEL
LIN {X 0,Y 86.685,Z 446.24,A -85,B 0,C 180,E1 -27284.074,E2 -27284.074} C_VEL
LIN {X 0,Y 89.251,Z 443.401,A -85,B 0,C 180,E1 -27290.751,E2 -27290.751} C_VEL
LIN {X 0,Y 91.511,Z 440.812,A -85,B 0,C 180,E1 -27294.983,E2 -27294.983} C_VEL
LIN {X 0,Y 95.763,Z 435.717,A -85,B 0,C 180,E1 -27300.91,E2 -27300.91} C_VEL
LIN {X 0,Y 99.959,Z 430.229,A -85,B 0,C 180,E1 -27305.451,E2 -27305.451} C_VEL
LIN {X 0,Y 104.729,Z 423.318,A -85,B 0,C 180,E1 -27309.604,E2 -27309.604} C_VEL
LIN {X 0,Y 109.263,Z 415.391,A -85,B 0,C 180,E1 -27313.109,E2 -27313.109} C_VEL
LIN {X 0,Y 113.126,Z 407.819,A -85,B 0,C 180,E1 -27315.594,E2 -27315.594} C_VEL
LIN {X 0,Y 116.622,Z 399.87,A -85,B 0,C 180,E1 -27317.577,E2 -27317.577} C_VEL
LIN {X 0,Y 119.484,Z 391.656,A -85,B 0,C 180,E1 -27319.224,E2 -27319.224} C_VEL
LIN {X 0,Y 121.788,Z 383.459,A -85,B 0,C 180,E1 -27320.475,E2 -27320.475} C_VEL
LIN {X 0,Y 123.63,Z 374.343,A -85,B 0,C 180,E1 -27321.554,E2 -27321.554} C_VEL
LIN {X 0,Y 124.879,Z 365.34,A -85,B 0,C 180,E1 -27322.269,E2 -27322.269} C_VEL
LIN {X 0,Y 125.555,Z 357.957,A -85,B 0,C 180,E1 -27322.678,E2 -27322.678} C_VEL
LIN {X 0,Y 121.391,Z 349.379,A -85,B 0,C 180,E1 -27326.268,E2 -27326.268} C_VEL
LIN {X 0,Y 117.715,Z 342.875,A -85,B 0,C 180,E1 -27329.866,E2 -27329.866} C_VEL
LIN {X 0,Y 114.158,Z 336.965,A -85,B 0,C 180,E1 -27333.982,E2 -27333.982} C_VEL
LIN {X 0,Y 111.247,Z 332.685,A -85,B 0,C 180,E1 -27338.03,E2 -27338.03} C_VEL
LIN {X 0,Y 108.893,Z 329.478,A -85,B 0,C 180,E1 -27342.086,E2 -27342.086} C_VEL
LIN {X 0,Y 108.257,Z 328.122,A -85,B 0,C 180,E1 -27343.499,E2 -27343.499} C_VEL
LIN {X 0,Y 105.952,Z 325.655,A -85,B 0,C 180,E1 -27349.489,E2 -27349.489} C_VEL
LIN {X 0,Y 105.109,Z 322.819,A -85,B 0,C 180,E1 -27354.243,E2 -27354.243} C_VEL
LIN {X 0,Y 104.687,Z 322.482,A -85,B 0,C 180,E1 -27360,E2 -27360} C_VEL
LIN {X 0,Y 105.137,Z 322.943,A -85,B 0,C 180,E1 -27365.273,E2 -27365.273} C_VEL
LIN {X 0,Y 106.763,Z 326.897,A -85,B 0,C 180,E1 -27372.353,E2 -27372.353} C_VEL
LIN {X 0,Y 108.459,Z 328.532,A -85,B 0,C 180,E1 -27376.227,E2 -27376.227} C_VEL
LIN {X 0,Y 110.818,Z 332.262,A -85,B 0,C 180,E1 -27380.596,E2 -27380.596} C_VEL
LIN {X 0,Y 112.022,Z 333.902,A -85,B 0,C 180,E1 -27382.416,E2 -27382.416} C_VEL
LIN {X 0,Y 114.807,Z 338.122,A -85,B 0,C 180,E1 -27386.111,E2 -27386.111} C_VEL
LIN {X 0,Y 117.498,Z 342.532,A -85,B 0,C 180,E1 -27389.175,E2 -27389.175} C_VEL
LIN {X 0,Y 119.358,Z 345.933,A -85,B 0,C 180,E1 -27391.101,E2 -27391.101} C_VEL
LIN {X 0,Y 122.781,Z 355.044,A -85,B 0,C 180,E1 -27394.543,E2 -27394.543} C_VEL
LIN {X 0,Y 124.436,Z 360.29,A -85,B 0,C 180,E1 -27396.123,E2 -27396.123} C_VEL
LIN {X 0,Y 124.685,Z 368.661,A -85,B 0,C 180,E1 -27397.061,E2 -27397.061} C_VEL
LIN {X 0,Y 123.098,Z 381.055,A -85,B 0,C 180,E1 -27397.839,E2 -27397.839} C_VEL
LIN {X 0,Y 121.022,Z 390.578,A -85,B 0,C 180,E1 -27398.761,E2 -27398.761} C_VEL
LIN {X 0,Y 118.828,Z 398.158,A -85,B 0,C 180,E1 -27399.75,E2 -27399.75} C_VEL
LIN {X 0,Y 115.654,Z 406.818,A -85,B 0,C 180,E1 -27401.24,E2 -27401.24} C_VEL
LIN {X 0,Y 112.036,Z 415.108,A -85,B 0,C 180,E1 -27403.181,E2 -27403.181} C_VEL
LIN {X 0,Y 108.473,Z 422.03,A -85,B 0,C 180,E1 -27405.266,E2 -27405.266} C_VEL
LIN {X 0,Y 104.658,Z 428.602,A -85,B 0,C 180,E1 -27407.819,E2 -27407.819} C_VEL
LIN {X 0,Y 100.6,Z 434.941,A -85,B 0,C 180,E1 -27411.045,E2 -27411.045} C_VEL
LIN {X 0,Y 96.802,Z 440.206,A -85,B 0,C 180,E1 -27414.495,E2 -27414.495} C_VEL
LIN {X 0,Y 93.534,Z 444.611,A -85,B 0,C 180,E1 -27418.269,E2 -27418.269} C_VEL
LIN {X 0,Y 89.338,Z 449.811,A -85,B 0,C 180,E1 -27424.365,E2 -27424.365} C_VEL
LIN {X 0,Y 86.379,Z 453.648,A -85,B 0,C 180,E1 -27431.01,E2 -27431.01} C_VEL
LIN {X 0,Y 85.087,Z 455.419,A -85,B 0,C 180,E1 -27435.656,E2 -27435.656} C_VEL
LIN {X 0,Y 84.339,Z 456.694,A -85,B 0,C 180,E1 -27440.409,E2 -27440.409} C_VEL
LIN {X 0,Y 84.071,Z 457.493,A -85,B 0,C 180,E1 -27445.207,E2 -27445.207} C_VEL
LIN {X 0,Y 84.257,Z 457.807,A -85,B 0,C 180,E1 -27450.002,E2 -27450.002} C_VEL
LIN {X 0,Y 84.074,Z 457.48,A -85,B 0,C 180,E1 -27454.798,E2 -27454.798} C_VEL
LIN {X 0,Y 84.34,Z 456.654,A -85,B 0,C 180,E1 -27459.596,E2 -27459.596} C_VEL
LIN {X 0,Y 85.087,Z 455.352,A -85,B 0,C 180,E1 -27464.349,E2 -27464.349} C_VEL
LIN {X 0,Y 87.238,Z 452.381,A -85,B 0,C 180,E1 -27471.258,E2 -27471.258} C_VEL
LIN {X 0,Y 89.339,Z 449.686,A -85,B 0,C 180,E1 -27475.639,E2 -27475.639} C_VEL
LIN {X 0,Y 93.532,Z 444.45,A -85,B 0,C 180,E1 -27481.737,E2 -27481.737} C_VEL
LIN {X 0,Y 98.646,Z 437.549,A -85,B 0,C 180,E1 -27487.273,E2 -27487.273} C_VEL
LIN {X 0,Y 103.631,Z 430.035,A -85,B 0,C 180,E1 -27491.395,E2 -27491.395} C_VEL
LIN {X 0,Y 107.84,Z 422.877,A -85,B 0,C 180,E1 -27494.317,E2 -27494.317} C_VEL
LIN {X 0,Y 111.403,Z 415.93,A -85,B 0,C 180,E1 -27496.512,E2 -27496.512} C_VEL
LIN {X 0,Y 115.009,Z 407.817,A -85,B 0,C 180,E1 -27498.469,E2 -27498.469} C_VEL
LIN {X 0,Y 118.141,Z 399.403,A -85,B 0,C 180,E1 -27499.99,E2 -27499.99} C_VEL
LIN {X 0,Y 120.935,Z 390.315,A -85,B 0,C 180,E1 -27501.147,E2 -27501.147} C_VEL
LIN {X 0,Y 123.337,Z 378.713,A -85,B 0,C 180,E1 -27502.257,E2 -27502.257} C_VEL
LIN {X 0,Y 124.463,Z 368.372,A -85,B 0,C 180,E1 -27502.88,E2 -27502.88} C_VEL
LIN {X 0,Y 124.132,Z 359.66,A -85,B 0,C 180,E1 -27503.901,E2 -27503.901} C_VEL
LIN {X 0,Y 120.978,Z 350.346,A -85,B 0,C 180,E1 -27506.939,E2 -27506.939} C_VEL
LIN {X 0,Y 118.346,Z 343.963,A -85,B 0,C 180,E1 -27509.653,E2 -27509.653} C_VEL
LIN {X 0,Y 114.071,Z 336.932,A -85,B 0,C 180,E1 -27514.452,E2 -27514.452} C_VEL
LIN {X 0,Y 111.012,Z 332.523,A -85,B 0,C 180,E1 -27518.653,E2 -27518.653} C_VEL
LIN {X 0,Y 108.71,Z 329.281,A -85,B 0,C 180,E1 -27522.603,E2 -27522.603} C_VEL
LIN {X 0,Y 108.076,Z 328.045,A -85,B 0,C 180,E1 -27523.962,E2 -27523.962} C_VEL
LIN {X 0,Y 105.866,Z 325.667,A -85,B 0,C 180,E1 -27529.481,E2 -27529.481} C_VEL
LIN {X 0,Y 105.002,Z 322.819,A -85,B 0,C 180,E1 -27533.756,E2 -27533.756} C_VEL
LIN {X 0,Y 104.35,Z 322.371,A -85,B 0,C 180,E1 -27540.441,E2 -27540.441} C_VEL
LIN {X 0,Y 104.386,Z 323.403,A -85,B 0,C 180,E1 -27543.608,E2 -27543.608} C_VEL
LIN {X 0,Y 104.562,Z 325.626,A -85,B 0,C 180,E1 -27546.613,E2 -27546.613} C_VEL
LIN {X 0,Y 106.054,Z 333.468,A -85,B 0,C 180,E1 -27554.222,E2 -27554.222} C_VEL
LIN {X 0,Y 106.806,Z 335.073,A -85,B 0,C 180,E1 -27556.173,E2 -27556.173} C_VEL
LIN {X 0,Y 108.878,Z 338.646,A -85,B 0,C 180,E1 -27560.349,E2 -27560.349} C_VEL
LIN {X 0,Y 109.948,Z 340.163,A -85,B 0,C 180,E1 -27562.098,E2 -27562.098} C_VEL
LIN {X 0,Y 112.504,Z 344.289,A -85,B 0,C 180,E1 -27565.775,E2 -27565.775} C_VEL
LIN {X 0,Y 115.734,Z 349.947,A -85,B 0,C 180,E1 -27569.674,E2 -27569.674} C_VEL
LIN {X 0,Y 119.627,Z 357.581,A -85,B 0,C 180,E1 -27573.675,E2 -27573.675} C_VEL
LIN {X 0,Y 120.887,Z 360.348,A -85,B 0,C 180,E1 -27574.86,E2 -27574.86} C_VEL
LIN {X 0,Y 119.552,Z 372.266,A -85,B 0,C 180,E1 -27575.711,E2 -27575.711} C_VEL
LIN {X 0,Y 117.848,Z 380.931,A -85,B 0,C 180,E1 -27576.61,E2 -27576.61} C_VEL
LIN {X 0,Y 115.081,Z 391.16,A -85,B 0,C 180,E1 -27578.159,E2 -27578.159} C_VEL
LIN {X 0,Y 111.974,Z 399.555,A -85,B 0,C 180,E1 -27579.745,E2 -27579.745} C_VEL
LIN {X 0,Y 108.327,Z 407.633,A -85,B 0,C 180,E1 -27581.744,E2 -27581.744} C_VEL
LIN {X 0,Y 104.256,Z 415.305,A -85,B 0,C 180,E1 -27584.252,E2 -27584.252} C_VEL
LIN {X 0,Y 99.428,Z 423.318,A -85,B 0,C 180,E1 -27587.814,E2 -27587.814} C_VEL
LIN {X 0,Y 94.365,Z 430.333,A -85,B 0,C 180,E1 -27592.086,E2 -27592.086} C_VEL
LIN {X 0,Y 89.814,Z 435.876,A -85,B 0,C 180,E1 -27596.784,E2 -27596.784} C_VEL
LIN {X 0,Y 85.173,Z 441.022,A -85,B 0,C 180,E1 -27603.008,E2 -27603.008} C_VEL
LIN {X 0,Y 82.673,Z 443.655,A -85,B 0,C 180,E1 -27607.506,E2 -27607.506} C_VEL
LIN {X 0,Y 79.886,Z 446.532,A -85,B 0,C 180,E1 -27614.694,E2 -27614.694} C_VEL
LIN {X 0,Y 78.254,Z 448.05,A -85,B 0,C 180,E1 -27621.084,E2 -27621.084} C_VEL
LIN {X 0,Y 77.437,Z 448.879,A -85,B 0,C 180,E1 -27629.997,E2 -27629.997} C_VEL
LIN {X 0,Y 78.253,Z 448.108,A -85,B 0,C 180,E1 -27638.911,E2 -27638.911} C_VEL
LIN {X 0,Y 79.824,Z 446.631,A -85,B 0,C 180,E1 -27645.313,E2 -27645.313} C_VEL
LIN {X 0,Y 82.661,Z 443.791,A -85,B 0,C 180,E1 -27652.492,E2 -27652.492} C_VEL
LIN {X 0,Y 85.143,Z 441.202,A -85,B 0,C 180,E1 -27656.997,E2 -27656.997} C_VEL
LIN {X 0,Y 89.773,Z 436.105,A -85,B 0,C 180,E1 -27663.227,E2 -27663.227} C_VEL
LIN {X 0,Y 94.286,Z 430.618,A -85,B 0,C 180,E1 -27667.945,E2 -27667.945} C_VEL
LIN {X 0,Y 99.372,Z 423.707,A -85,B 0,C 180,E1 -27672.209,E2 -27672.209} C_VEL
LIN {X 0,Y 104.211,Z 415.778,A -85,B 0,C 180,E1 -27675.767,E2 -27675.767} C_VEL
LIN {X 0,Y 108.285,Z 408.206,A -85,B 0,C 180,E1 -27678.275,E2 -27678.275} C_VEL
LIN {X 0,Y 111.977,Z 400.255,A -85,B 0,C 180,E1 -27680.247,E2 -27680.247} C_VEL
LIN {X 0,Y 114.991,Z 392.041,A -85,B 0,C 180,E1 -27681.892,E2 -27681.892} C_VEL
LIN {X 0,Y 117.454,Z 383.71,A -85,B 0,C 180,E1 -27683.15,E2 -27683.15} C_VEL
LIN {X 0,Y 119.41,Z 374.451,A -85,B 0,C 180,E1 -27684.24,E2 -27684.24} C_VEL
LIN {X 0,Y 120.724,Z 365.355,A -85,B 0,C 180,E1 -27684.946,E2 -27684.946} C_VEL
LIN {X 0,Y 121.171,Z 360.817,A -85,B 0,C 180,E1 -27685.233,E2 -27685.233} C_VEL
LIN {X 0,Y 117.599,Z 353.298,A -85,B 0,C 180,E1 -27688.729,E2 -27688.729} C_VEL
LIN {X 0,Y 114.292,Z 347.087,A -85,B 0,C 180,E1 -27692.446,E2 -27692.446} C_VEL
LIN {X 0,Y 111.484,Z 342.452,A -85,B 0,C 180,E1 -27696.129,E2 -27696.129} C_VEL
LIN {X 0,Y 109.347,Z 339.035,A -85,B 0,C 180,E1 -27699.482,E2 -27699.482} C_VEL
LIN {X 0,Y 107.14,Z 335.549,A -85,B 0,C 180,E1 -27703.812,E2 -27703.812} C_VEL
LIN {X 0,Y 106.76,Z 334.824,A -85,B 0,C 180,E1 -27704.732,E2 -27704.732} C_VEL
LIN {X 0,Y 104.723,Z 332.225,A -85,B 0,C 180,E1 -27710.828,E2 -27710.828} C_VEL
LIN {X 0,Y 104.103,Z 329.811,A -85,B 0,C 180,E1 -27715.159,E2 -27715.159} C_VEL
LIN {X 0,Y 103.824,Z 329.51,A -85,B 0,C 180,E1 -27720,E2 -27720} C_VEL
LIN {X 0,Y 104.177,Z 330.038,A -85,B 0,C 180,E1 -27724.776,E2 -27724.776} C_VEL
LIN {X 0,Y 105.77,Z 333.974,A -85,B 0,C 180,E1 -27732.106,E2 -27732.106} C_VEL
LIN {X 0,Y 107,Z 335.227,A -85,B 0,C 180,E1 -27735.11,E2 -27735.11} C_VEL
LIN {X 0,Y 109.445,Z 339.145,A -85,B 0,C 180,E1 -27739.946,E2 -27739.946} C_VEL
LIN {X 0,Y 112.673,Z 344.367,A -85,B 0,C 180,E1 -27744.776,E2 -27744.776} C_VEL
LIN {X 0,Y 115.937,Z 350.045,A -85,B 0,C 180,E1 -27748.736,E2 -27748.736} C_VEL
LIN {X 0,Y 119.265,Z 359.471,A -85,B 0,C 180,E1 -27752.528,E2 -27752.528} C_VEL
LIN {X 0,Y 120.341,Z 363.16,A -85,B 0,C 180,E1 -27753.699,E2 -27753.699} C_VEL
LIN {X 0,Y 120.302,Z 370.927,A -85,B 0,C 180,E1 -27754.525,E2 -27754.525} C_VEL
LIN {X 0,Y 118.744,Z 381.341,A -85,B 0,C 180,E1 -27755.193,E2 -27755.193} C_VEL
LIN {X 0,Y 116.508,Z 390.948,A -85,B 0,C 180,E1 -27756.136,E2 -27756.136} C_VEL
LIN {X 0,Y 113.747,Z 399.647,A -85,B 0,C 180,E1 -27757.301,E2 -27757.301} C_VEL
LIN {X 0,Y 110.459,Z 407.935,A -85,B 0,C 180,E1 -27758.796,E2 -27758.796} C_VEL
LIN {X 0,Y 106.035,Z 417.183,A -85,B 0,C 180,E1 -27761.071,E2 -27761.071} C_VEL
LIN {X 0,Y 100.517,Z 426.663,A -85,B 0,C 180,E1 -27764.361,E2 -27764.361} C_VEL
LIN {X 0,Y 96.241,Z 433.123,A -85,B 0,C 180,E1 -27767.512,E2 -27767.512} C_VEL
LIN {X 0,Y 92.084,Z 438.635,A -85,B 0,C 180,E1 -27770.979,E2 -27770.979} C_VEL
LIN {X 0,Y 87.577,Z 444.221,A -85,B 0,C 180,E1 -27775.826,E2 -27775.826} C_VEL
LIN {X 0,Y 82.963,Z 449.419,A -85,B 0,C 180,E1 -27782.233,E2 -27782.233} C_VEL
LIN {X 0,Y 79.678,Z 453.256,A -85,B 0,C 180,E1 -27789.343,E2 -27789.343} C_VEL
LIN {X 0,Y 78.206,Z 455.026,A -85,B 0,C 180,E1 -27794.363,E2 -27794.363} C_VEL
LIN {X 0,Y 77.315,Z 456.301,A -85,B 0,C 180,E1 -27799.528,E2 -27799.528} C_VEL
LIN {X 0,Y 76.991,Z 457.101,A -85,B 0,C 180,E1 -27804.765,E2 -27804.765} C_VEL
LIN {X 0,Y 77.16,Z 457.415,A -85,B 0,C 180,E1 -27810.003,E2 -27810.003} C_VEL
LIN {X 0,Y 76.993,Z 457.087,A -85,B 0,C 180,E1 -27815.24,E2 -27815.24} C_VEL
LIN {X 0,Y 77.316,Z 456.26,A -85,B 0,C 180,E1 -27820.477,E2 -27820.477} C_VEL
LIN {X 0,Y 78.206,Z 454.958,A -85,B 0,C 180,E1 -27825.643,E2 -27825.643} C_VEL
LIN {X 0,Y 80.62,Z 451.986,A -85,B 0,C 180,E1 -27833.099,E2 -27833.099} C_VEL
LIN {X 0,Y 82.965,Z 449.291,A -85,B 0,C 180,E1 -27837.772,E2 -27837.772} C_VEL
LIN {X 0,Y 87.575,Z 444.056,A -85,B 0,C 180,E1 -27844.18,E2 -27844.18} C_VEL
LIN {X 0,Y 93.101,Z 437.156,A -85,B 0,C 180,E1 -27849.917,E2 -27849.917} C_VEL
LIN {X 0,Y 98.401,Z 429.639,A -85,B 0,C 180,E1 -27854.139,E2 -27854.139} C_VEL
LIN {X 0,Y 102.419,Z 423.26,A -85,B 0,C 180,E1 -27856.811,E2 -27856.811} C_VEL
LIN {X 0,Y 106.628,Z 415.533,A -85,B 0,C 180,E1 -27859.289,E2 -27859.289} C_VEL
LIN {X 0,Y 110.442,Z 407.422,A -85,B 0,C 180,E1 -27861.22,E2 -27861.22} C_VEL
LIN {X 0,Y 113.722,Z 399.006,A -85,B 0,C 180,E1 -27862.722,E2 -27862.722} C_VEL
LIN {X 0,Y 116.73,Z 389.423,A -85,B 0,C 180,E1 -27863.933,E2 -27863.933} C_VEL
LIN {X 0,Y 119.206,Z 377.755,A -85,B 0,C 180,E1 -27865.002,E2 -27865.002} C_VEL
LIN {X 0,Y 120.201,Z 368.883,A -85,B 0,C 180,E1 -27865.558,E2 -27865.558} C_VEL
LIN {X 0,Y 120.058,Z 362.625,A -85,B 0,C 180,E1 -27866.304,E2 -27866.304} C_VEL
LIN {X 0,Y 117.228,Z 353.858,A -85,B 0,C 180,E1 -27869.411,E2 -27869.411} C_VEL
LIN {X 0,Y 115.359,Z 349.176,A -85,B 0,C 180,E1 -27871.579,E2 -27871.579} C_VEL
LIN {X 0,Y 111.708,Z 342.858,A -85,B 0,C 180,E1 -27876.14,E2 -27876.14} C_VEL
LIN {X 0,Y 109.168,Z 338.944,A -85,B 0,C 180,E1 -27880.001,E2 -27880.001} C_VEL
LIN {X 0,Y 106.894,Z 335.223,A -85,B 0,C 180,E1 -27884.448,E2 -27884.448} C_VEL
LIN {X 0,Y 104.419,Z 331.715,A -85,B 0,C 180,E1 -27891.656,E2 -27891.656} C_VEL
LIN {X 0,Y 103.92,Z 329.772,A -85,B 0,C 180,E1 -27894.908,E2 -27894.908} C_VEL
LIN {X 0,Y 103.509,Z 329.522,A -85,B 0,C 180,E1 -27901.946,E2 -27901.946} C_VEL
LIN {X 0,Y 103.973,Z 329.919,A -85,B 0,C 180,E1 -27906.307,E2 -27906.307} C_VEL
LIN {X 0,Y 105.29,Z 333.495,A -85,B 0,C 180,E1 -27912.424,E2 -27912.424} C_VEL
LIN {X 0,Y 106.806,Z 335.073,A -85,B 0,C 180,E1 -27916.173,E2 -27916.173} C_VEL
LIN {X 0,Y 107.993,Z 337.893,A -85,B 0,C 180,E1 -27918.858,E2 -27918.858} C_VEL
LIN {X 0,Y 109.053,Z 341.764,A -85,B 0,C 180,E1 -27921.176,E2 -27921.176} C_VEL
LIN {X 0,Y 112.138,Z 353.479,A -85,B 0,C 180,E1 -27926.711,E2 -27926.711} C_VEL
LIN {X 0,Y 113.289,Z 356.002,A -85,B 0,C 180,E1 -27928.203,E2 -27928.203} C_VEL
LIN {X 0,Y 116.482,Z 362.755,A -85,B 0,C 180,E1 -27931.855,E2 -27931.855} C_VEL
LIN {X 0,Y 116.76,Z 363.492,A -85,B 0,C 180,E1 -27932.193,E2 -27932.193} C_VEL
LIN {X 0,Y 115.42,Z 373.344,A -85,B 0,C 180,E1 -27932.914,E2 -27932.914} C_VEL
LIN {X 0,Y 113.646,Z 381.827,A -85,B 0,C 180,E1 -27933.819,E2 -27933.819} C_VEL
LIN {X 0,Y 111.479,Z 389.693,A -85,B 0,C 180,E1 -27934.956,E2 -27934.956} C_VEL
LIN {X 0,Y 108.277,Z 398.452,A -85,B 0,C 180,E1 -27936.557,E2 -27936.557} C_VEL
LIN {X 0,Y 104.375,Z 406.803,A -85,B 0,C 180,E1 -27938.483,E2 -27938.483} C_VEL
LIN {X 0,Y 100.087,Z 414.679,A -85,B 0,C 180,E1 -27940.985,E2 -27940.985} C_VEL
LIN {X 0,Y 96.54,Z 420.332,A -85,B 0,C 180,E1 -27943.279,E2 -27943.279} C_VEL
LIN {X 0,Y 92.077,Z 426.643,A -85,B 0,C 180,E1 -27946.609,E2 -27946.609} C_VEL
LIN {X 0,Y 87.866,Z 431.89,A -85,B 0,C 180,E1 -27950.214,E2 -27950.214} C_VEL
LIN {X 0,Y 83.994,Z 436.267,A -85,B 0,C 180,E1 -27954.144,E2 -27954.144} C_VEL
LIN {X 0,Y 78.93,Z 441.414,A -85,B 0,C 180,E1 -27960.675,E2 -27960.675} C_VEL
LIN {X 0,Y 76.185,Z 444.046,A -85,B 0,C 180,E1 -27965.47,E2 -27965.47} C_VEL
LIN {X 0,Y 73.068,Z 446.924,A -85,B 0,C 180,E1 -27973.226,E2 -27973.226} C_VEL
LIN {X 0,Y 71.016,Z 448.704,A -85,B 0,C 180,E1 -27981.747,E2 -27981.747} C_VEL
LIN {X 0,Y 70.369,Z 449.27,A -85,B 0,C 180,E1 -27989.997,E2 -27989.997} C_VEL
LIN {X 0,Y 70.937,Z 448.825,A -85,B 0,C 180,E1 -27997.801,E2 -27997.801} C_VEL
LIN {X 0,Y 73.033,Z 447.021,A -85,B 0,C 180,E1 -28006.776,E2 -28006.776} C_VEL
LIN {X 0,Y 76.173,Z 444.181,A -85,B 0,C 180,E1 -28014.528,E2 -28014.528} C_VEL
LIN {X 0,Y 78.905,Z 441.592,A -85,B 0,C 180,E1 -28019.329,E2 -28019.329} C_VEL
LIN {X 0,Y 83.95,Z 436.494,A -85,B 0,C 180,E1 -28025.872,E2 -28025.872} C_VEL
LIN {X 0,Y 88.813,Z 431.007,A -85,B 0,C 180,E1 -28030.753,E2 -28030.753} C_VEL
LIN {X 0,Y 94.248,Z 424.095,A -85,B 0,C 180,E1 -28035.102,E2 -28035.102} C_VEL
LIN {X 0,Y 99.41,Z 416.165,A -85,B 0,C 180,E1 -28038.687,E2 -28038.687} C_VEL
LIN {X 0,Y 103.704,Z 408.594,A -85,B 0,C 180,E1 -28041.198,E2 -28041.198} C_VEL
LIN {X 0,Y 107.593,Z 400.64,A -85,B 0,C 180,E1 -28043.143,E2 -28043.143} C_VEL
LIN {X 0,Y 110.764,Z 392.425,A -85,B 0,C 180,E1 -28044.774,E2 -28044.774} C_VEL
LIN {X 0,Y 113.392,Z 383.938,A -85,B 0,C 180,E1 -28046.035,E2 -28046.035} C_VEL
LIN {X 0,Y 115.502,Z 374.451,A -85,B 0,C 180,E1 -28047.119,E2 -28047.119} C_VEL
LIN {X 0,Y 116.938,Z 364.752,A -85,B 0,C 180,E1 -28047.837,E2 -28047.837} C_VEL
LIN {X 0,Y 116.915,Z 363.531,A -85,B 0,C 180,E1 -28048.049,E2 -28048.049} C_VEL
LIN {X 0,Y 113.493,Z 356.083,A -85,B 0,C 180,E1 -28052.014,E2 -28052.014} C_VEL
LIN {X 0,Y 110.83,Z 351.046,A -85,B 0,C 180,E1 -28055.545,E2 -28055.545} C_VEL
LIN {X 0,Y 109.007,Z 347.937,A -85,B 0,C 180,E1 -28058.333,E2 -28058.333} C_VEL
LIN {X 0,Y 107.551,Z 345.407,A -85,B 0,C 180,E1 -28060.929,E2 -28060.929} C_VEL
LIN {X 0,Y 105.432,Z 341.627,A -85,B 0,C 180,E1 -28065.711,E2 -28065.711} C_VEL
LIN {X 0,Y 103.594,Z 338.929,A -85,B 0,C 180,E1 -28071.956,E2 -28071.956} C_VEL
LIN {X 0,Y 103.178,Z 336.832,A -85,B 0,C 180,E1 -28075.605,E2 -28075.605} C_VEL
LIN {X 0,Y 102.958,Z 336.565,A -85,B 0,C 180,E1 -28080,E2 -28080} C_VEL
LIN {X 0,Y 103.218,Z 337.111,A -85,B 0,C 180,E1 -28084.209,E2 -28084.209} C_VEL
LIN {X 0,Y 104.623,Z 340.833,A -85,B 0,C 180,E1 -28091.38,E2 -28091.38} C_VEL
LIN {X 0,Y 105.671,Z 342.104,A -85,B 0,C 180,E1 -28094.196,E2 -28094.196} C_VEL
LIN {X 0,Y 108.297,Z 346.621,A -85,B 0,C 180,E1 -28099.703,E2 -28099.703} C_VEL
LIN {X 0,Y 110.751,Z 350.936,A -85,B 0,C 180,E1 -28103.614,E2 -28103.614} C_VEL
LIN {X 0,Y 113.346,Z 355.83,A -85,B 0,C 180,E1 -28107.078,E2 -28107.078} C_VEL
LIN {X 0,Y 116.105,Z 364.79,A -85,B 0,C 180,E1 -28110.663,E2 -28110.663} C_VEL
LIN {X 0,Y 116.476,Z 366.197,A -85,B 0,C 180,E1 -28111.129,E2 -28111.129} C_VEL
LIN {X 0,Y 116.2,Z 372.254,A -85,B 0,C 180,E1 -28111.735,E2 -28111.735} C_VEL
LIN {X 0,Y 114.569,Z 382.024,A -85,B 0,C 180,E1 -28112.377,E2 -28112.377} C_VEL
LIN {X 0,Y 112.241,Z 391.375,A -85,B 0,C 180,E1 -28113.31,E2 -28113.31} C_VEL
LIN {X 0,Y 108.895,Z 401.137,A -85,B 0,C 180,E1 -28114.63,E2 -28114.63} C_VEL
LIN {X 0,Y 104.133,Z 411.864,A -85,B 0,C 180,E1 -28116.735,E2 -28116.735} C_VEL
LIN {X 0,Y 99.567,Z 420.133,A -85,B 0,C 180,E1 -28119.068,E2 -28119.068} C_VEL
LIN {X 0,Y 94.595,Z 427.821,A -85,B 0,C 180,E1 -28122.019,E2 -28122.019} C_VEL
LIN {X 0,Y 89.986,Z 434.16,A -85,B 0,C 180,E1 -28125.343,E2 -28125.343} C_VEL
LIN {X 0,Y 85.622,Z 439.425,A -85,B 0,C 180,E1 -28128.958,E2 -28128.958} C_VEL
LIN {X 0,Y 81.786,Z 443.829,A -85,B 0,C 180,E1 -28133.024,E2 -28133.024} C_VEL
LIN {X 0,Y 76.73,Z 449.027,A -85,B 0,C 180,E1 -28139.754,E2 -28139.754} C_VEL
LIN {X 0,Y 73.059,Z 452.864,A -85,B 0,C 180,E1 -28147.373,E2 -28147.373} C_VEL
LIN {X 0,Y 71.383,Z 454.634,A -85,B 0,C 180,E1 -28152.824,E2 -28152.824} C_VEL
LIN {X 0,Y 70.329,Z 455.909,A -85,B 0,C 180,E1 -28158.474,E2 -28158.474} C_VEL
LIN {X 0,Y 69.909,Z 456.708,A -85,B 0,C 180,E1 -28164.233,E2 -28164.233} C_VEL
LIN {X 0,Y 70.074,Z 457.024,A -85,B 0,C 180,E1 -28170.003,E2 -28170.003} C_VEL
LIN {X 0,Y 69.91,Z 456.694,A -85,B 0,C 180,E1 -28175.773,E2 -28175.773} C_VEL
LIN {X 0,Y 70.33,Z 455.867,A -85,B 0,C 180,E1 -28181.532,E2 -28181.532} C_VEL
LIN {X 0,Y 71.383,Z 454.564,A -85,B 0,C 180,E1 -28187.182,E2 -28187.182} C_VEL
LIN {X 0,Y 74.11,Z 451.591,A -85,B 0,C 180,E1 -28195.264,E2 -28195.264} C_VEL
LIN {X 0,Y 76.732,Z 448.896,A -85,B 0,C 180,E1 -28200.252,E2 -28200.252} C_VEL
LIN {X 0,Y 81.784,Z 443.662,A -85,B 0,C 180,E1 -28206.983,E2 -28206.983} C_VEL
LIN {X 0,Y 86.683,Z 438.037,A -85,B 0,C 180,E1 -28211.984,E2 -28211.984} C_VEL
LIN {X 0,Y 92.804,Z 430.14,A -85,B 0,C 180,E1 -28216.758,E2 -28216.758} C_VEL
LIN {X 0,Y 97.699,Z 422.865,A -85,B 0,C 180,E1 -28219.846,E2 -28219.846} C_VEL
LIN {X 0,Y 102.129,Z 415.136,A -85,B 0,C 180,E1 -28222.317,E2 -28222.317} C_VEL
LIN {X 0,Y 106.141,Z 407.025,A -85,B 0,C 180,E1 -28224.208,E2 -28224.208} C_VEL
LIN {X 0,Y 109.568,Z 398.608,A -85,B 0,C 180,E1 -28225.676,E2 -28225.676} C_VEL
LIN {X 0,Y 112.706,Z 389.024,A -85,B 0,C 180,E1 -28226.844,E2 -28226.844} C_VEL
LIN {X 0,Y 115.24,Z 377.53,A -85,B 0,C 180,E1 -28227.891,E2 -28227.891} C_VEL
LIN {X 0,Y 116.21,Z 369.838,A -85,B 0,C 180,E1 -28228.358,E2 -28228.358} C_VEL
LIN {X 0,Y 116.144,Z 365.419,A -85,B 0,C 180,E1 -28228.944,E2 -28228.944} C_VEL
LIN {X 0,Y 113.22,Z 355.944,A -85,B 0,C 180,E1 -28232.693,E2 -28232.693} C_VEL
LIN {X 0,Y 110.497,Z 350.641,A -85,B 0,C 180,E1 -28236.329,E2 -28236.329} C_VEL
LIN {X 0,Y 107.516,Z 345.49,A -85,B 0,C 180,E1 -28241.171,E2 -28241.171} C_VEL
LIN {X 0,Y 105.27,Z 341.544,A -85,B 0,C 180,E1 -28246.084,E2 -28246.084} C_VEL
LIN {X 0,Y 103.457,Z 338.96,A -85,B 0,C 180,E1 -28251.885,E2 -28251.885} C_VEL
LIN {X 0,Y 102.961,Z 336.792,A -85,B 0,C 180,E1 -28255.474,E2 -28255.474} C_VEL
LIN {X 0,Y 102.644,Z 336.572,A -85,B 0,C 180,E1 -28261.962,E2 -28261.962} C_VEL
LIN {X 0,Y 102.985,Z 336.965,A -85,B 0,C 180,E1 -28265.63,E2 -28265.63} C_VEL
LIN {X 0,Y 104.228,Z 340.464,A -85,B 0,C 180,E1 -28271.93,E2 -28271.93} C_VEL
LIN {X 0,Y 105.379,Z 341.785,A -85,B 0,C 180,E1 -28275.033,E2 -28275.033} C_VEL
LIN {X 0,Y 107.517,Z 345.498,A -85,B 0,C 180,E1 -28279.653,E2 -28279.653} C_VEL
LIN {X 0,Y 110.245,Z 350.192,A -85,B 0,C 180,E1 -28284.128,E2 -28284.128} C_VEL
LIN {X 0,Y 113.289,Z 356.002,A -85,B 0,C 180,E1 -28288.203,E2 -28288.203} C_VEL
LIN {X 0,Y 114.265,Z 358.775,A -85,B 0,C 180,E1 -28289.461,E2 -28289.461} C_VEL
LIN {X 0,Y 114.732,Z 362.245,A -85,B 0,C 180,E1 -28290.318,E2 -28290.318} C_VEL
LIN {X 0,Y 114.697,Z 366.089,A -85,B 0,C 180,E1 -28290.85,E2 -28290.85} C_VEL
LIN {X 0,Y 114.123,Z 370.009,A -85,B 0,C 180,E1 -28291.084,E2 -28291.084} C_VEL
LIN {X 0,Y 110.679,Z 380.642,A -85,B 0,C 180,E1 -28290.893,E2 -28290.893} C_VEL
LIN {X 0,Y 108.607,Z 386.905,A -85,B 0,C 180,E1 -28291.392,E2 -28291.392} C_VEL
LIN {X 0,Y 104.886,Z 397.352,A -85,B 0,C 180,E1 -28293.112,E2 -28293.112} C_VEL
LIN {X 0,Y 100.8,Z 405.972,A -85,B 0,C 180,E1 -28294.988,E2 -28294.988} C_VEL
LIN {X 0,Y 96.232,Z 414.058,A -85,B 0,C 180,E1 -28297.415,E2 -28297.415} C_VEL
LIN {X 0,Y 91.823,Z 420.727,A -85,B 0,C 180,E1 -28300.056,E2 -28300.056} C_VEL
LIN {X 0,Y 87.075,Z 427.036,A -85,B 0,C 180,E1 -28303.411,E2 -28303.411} C_VEL
LIN {X 0,Y 82.54,Z 432.283,A -85,B 0,C 180,E1 -28307.062,E2 -28307.062} C_VEL
LIN {X 0,Y 78.378,Z 436.659,A -85,B 0,C 180,E1 -28311.118,E2 -28311.118} C_VEL
LIN {X 0,Y 72.849,Z 441.806,A -85,B 0,C 180,E1 -28317.95,E2 -28317.95} C_VEL
LIN {X 0,Y 69.804,Z 444.438,A -85,B 0,C 180,E1 -28323.056,E2 -28323.056} C_VEL
LIN {X 0,Y 66.317,Z 447.316,A -85,B 0,C 180,E1 -28331.459,E2 -28331.459} C_VEL
LIN {X 0,Y 64.655,Z 448.571,A -85,B 0,C 180,E1 -28337.44,E2 -28337.44} C_VEL
LIN {X 0,Y 63.642,Z 449.359,A -85,B 0,C 180,E1 -28343.657,E2 -28343.657} C_VEL
LIN {X 0,Y 63.293,Z 449.66,A -85,B 0,C 180,E1 -28349.997,E2 -28349.997} C_VEL
LIN {X 0,Y 63.642,Z 449.378,A -85,B 0,C 180,E1 -28356.337,E2 -28356.337} C_VEL
LIN {X 0,Y 64.653,Z 448.627,A -85,B 0,C 180,E1 -28362.553,E2 -28362.553} C_VEL
LIN {X 0,Y 66.279,Z 447.411,A -85,B 0,C 180,E1 -28368.545,E2 -28368.545} C_VEL
LIN {X 0,Y 69.792,Z 444.571,A -85,B 0,C 180,E1 -28376.942,E2 -28376.942} C_VEL
LIN {X 0,Y 72.824,Z 441.981,A -85,B 0,C 180,E1 -28382.055,E2 -28382.055} C_VEL
LIN {X 0,Y 78.331,Z 436.883,A -85,B 0,C 180,E1 -28388.903,E2 -28388.903} C_VEL
LIN {X 0,Y 83.583,Z 431.396,A -85,B 0,C 180,E1 -28393.92,E2 -28393.92} C_VEL
LIN {X 0,Y 89.392,Z 424.483,A -85,B 0,C 180,E1 -28398.318,E2 -28398.318} C_VEL
LIN {X 0,Y 94.886,Z 416.553,A -85,B 0,C 180,E1 -28401.9,E2 -28401.9} C_VEL
LIN {X 0,Y 99.42,Z 408.981,A -85,B 0,C 180,E1 -28404.38,E2 -28404.38} C_VEL
LIN {X 0,Y 102.825,Z 402.522,A -85,B 0,C 180,E1 -28405.965,E2 -28405.965} C_VEL
LIN {X 0,Y 106.185,Z 394.674,A -85,B 0,C 180,E1 -28407.548,E2 -28407.548} C_VEL
LIN {X 0,Y 109.288,Z 385.385,A -85,B 0,C 180,E1 -28408.978,E2 -28408.978} C_VEL
LIN {X 0,Y 111.624,Z 375.728,A -85,B 0,C 180,E1 -28410.094,E2 -28410.094} C_VEL
LIN {X 0,Y 113.037,Z 366.798,A -85,B 0,C 180,E1 -28410.839,E2 -28410.839} C_VEL
LIN {X 0,Y 110.318,Z 360.39,A -85,B 0,C 180,E1 -28414.694,E2 -28414.694} C_VEL
LIN {X 0,Y 107.775,Z 355.255,A -85,B 0,C 180,E1 -28418.7,E2 -28418.7} C_VEL
LIN {X 0,Y 105.801,Z 351.72,A -85,B 0,C 180,E1 -28422.482,E2 -28422.482} C_VEL
LIN {X 0,Y 104.024,Z 348.311,A -85,B 0,C 180,E1 -28427.022,E2 -28427.022} C_VEL
LIN {X 0,Y 102.438,Z 345.317,A -85,B 0,C 180,E1 -28433.66,E2 -28433.66} C_VEL
LIN {X 0,Y 102.248,Z 343.949,A -85,B 0,C 180,E1 -28436.058,E2 -28436.058} C_VEL
LIN {X 0,Y 102.094,Z 343.6,A -85,B 0,C 180,E1 -28440,E2 -28440} C_VEL
LIN {X 0,Y 102.263,Z 344.051,A -85,B 0,C 180,E1 -28443.447,E2 -28443.447} C_VEL
LIN {X 0,Y 103.455,Z 347.662,A -85,B 0,C 180,E1 -28450.519,E2 -28450.519} C_VEL
LIN {X 0,Y 104.3,Z 348.805,A -85,B 0,C 180,E1 -28453.052,E2 -28453.052} C_VEL
LIN {X 0,Y 106.638,Z 353.193,A -85,B 0,C 180,E1 -28458.491,E2 -28458.491} C_VEL
LIN {X 0,Y 108.883,Z 357.439,A -85,B 0,C 180,E1 -28462.409,E2 -28462.409} C_VEL
LIN {X 0,Y 110.768,Z 361.487,A -85,B 0,C 180,E1 -28465.232,E2 -28465.232} C_VEL
LIN {X 0,Y 112.815,Z 369.01,A -85,B 0,C 180,E1 -28468.328,E2 -28468.328} C_VEL
LIN {X 0,Y 112.466,Z 373.055,A -85,B 0,C 180,E1 -28468.723,E2 -28468.723} C_VEL
LIN {X 0,Y 110.782,Z 382.358,A -85,B 0,C 180,E1 -28469.342,E2 -28469.342} C_VEL
LIN {X 0,Y 108.079,Z 392.418,A -85,B 0,C 180,E1 -28470.333,E2 -28470.333} C_VEL
LIN {X 0,Y 103.581,Z 404.153,A -85,B 0,C 180,E1 -28471.996,E2 -28471.996} C_VEL
LIN {X 0,Y 99.354,Z 412.708,A -85,B 0,C 180,E1 -28473.786,E2 -28473.786} C_VEL
LIN {X 0,Y 94.575,Z 420.768,A -85,B 0,C 180,E1 -28476.09,E2 -28476.09} C_VEL
LIN {X 0,Y 89.999,Z 427.432,A -85,B 0,C 180,E1 -28478.661,E2 -28478.661} C_VEL
LIN {X 0,Y 85.073,Z 433.77,A -85,B 0,C 180,E1 -28481.973,E2 -28481.973} C_VEL
LIN {X 0,Y 80.401,Z 439.035,A -85,B 0,C 180,E1 -28485.633,E2 -28485.633} C_VEL
LIN {X 0,Y 76.201,Z 443.436,A -85,B 0,C 180,E1 -28489.793,E2 -28489.793} C_VEL
LIN {X 0,Y 70.673,Z 448.635,A -85,B 0,C 180,E1 -28496.846,E2 -28496.846} C_VEL
LIN {X 0,Y 66.529,Z 452.471,A -85,B 0,C 180,E1 -28505.008,E2 -28505.008} C_VEL
LIN {X 0,Y 64.601,Z 454.241,A -85,B 0,C 180,E1 -28510.955,E2 -28510.955} C_VEL
LIN {X 0,Y 63.361,Z 455.515,A -85,B 0,C 180,E1 -28517.186,E2 -28517.186} C_VEL
LIN {X 0,Y 62.839,Z 456.316,A -85,B 0,C 180,E1 -28523.582,E2 -28523.582} C_VEL
LIN {X 0,Y 62.99,Z 456.633,A -85,B 0,C 180,E1 -28530.003,E2 -28530.003} C_VEL
LIN {X 0,Y 62.841,Z 456.302,A -85,B 0,C 180,E1 -28536.425,E2 -28536.425} C_VEL
LIN {X 0,Y 63.362,Z 455.473,A -85,B 0,C 180,E1 -28542.82,E2 -28542.82} C_VEL
LIN {X 0,Y 64.601,Z 454.17,A -85,B 0,C 180,E1 -28549.052,E2 -28549.052} C_VEL
LIN {X 0,Y 67.734,Z 451.197,A -85,B 0,C 180,E1 -28557.838,E2 -28557.838} C_VEL
LIN {X 0,Y 70.675,Z 448.502,A -85,B 0,C 180,E1 -28563.16,E2 -28563.16} C_VEL
LIN {X 0,Y 76.198,Z 443.266,A -85,B 0,C 180,E1 -28570.216,E2 -28570.216} C_VEL
LIN {X 0,Y 81.549,Z 437.644,A -85,B 0,C 180,E1 -28575.319,E2 -28575.319} C_VEL
LIN {X 0,Y 88.066,Z 429.755,A -85,B 0,C 180,E1 -28580.132,E2 -28580.132} C_VEL
LIN {X 0,Y 93.279,Z 422.47,A -85,B 0,C 180,E1 -28583.181,E2 -28583.181} C_VEL
LIN {X 0,Y 97.947,Z 414.74,A -85,B 0,C 180,E1 -28585.608,E2 -28585.608} C_VEL
LIN {X 0,Y 102.14,Z 406.627,A -85,B 0,C 180,E1 -28587.45,E2 -28587.45} C_VEL
LIN {X 0,Y 105.736,Z 398.211,A -85,B 0,C 180,E1 -28588.848,E2 -28588.848} C_VEL
LIN {X 0,Y 109.137,Z 388.098,A -85,B 0,C 180,E1 -28590.033,E2 -28590.033} C_VEL
LIN {X 0,Y 111.908,Z 375.198,A -85,B 0,C 180,E1 -28591.087,E2 -28591.087} C_VEL
LIN {X 0,Y 112.502,Z 370.057,A -85,B 0,C 180,E1 -28591.455,E2 -28591.455} C_VEL
LIN {X 0,Y 112.434,Z 368.041,A -85,B 0,C 180,E1 -28591.84,E2 -28591.84} C_VEL
LIN {X 0,Y 110.3,Z 360.611,A -85,B 0,C 180,E1 -28595.032,E2 -28595.032} C_VEL
LIN {X 0,Y 107.677,Z 355.308,A -85,B 0,C 180,E1 -28599.088,E2 -28599.088} C_VEL
LIN {X 0,Y 105.594,Z 351.6,A -85,B 0,C 180,E1 -28603.009,E2 -28603.009} C_VEL
LIN {X 0,Y 103.956,Z 348.308,A -85,B 0,C 180,E1 -28607.105,E2 -28607.105} C_VEL
LIN {X 0,Y 102.29,Z 345.478,A -85,B 0,C 180,E1 -28613.342,E2 -28613.342} C_VEL
LIN {X 0,Y 102.01,Z 343.835,A -85,B 0,C 180,E1 -28616.05,E2 -28616.05} C_VEL
LIN {X 0,Y 101.779,Z 343.618,A -85,B 0,C 180,E1 -28621.979,E2 -28621.979} C_VEL
LIN {X 0,Y 102.014,Z 343.99,A -85,B 0,C 180,E1 -28624.941,E2 -28624.941} C_VEL
LIN {X 0,Y 103.11,Z 347.357,A -85,B 0,C 180,E1 -28631.215,E2 -28631.215} C_VEL
LIN {X 0,Y 104.056,Z 348.642,A -85,B 0,C 180,E1 -28634.044,E2 -28634.044} C_VEL
LIN {X 0,Y 106.42,Z 353.051,A -85,B 0,C 180,E1 -28639.476,E2 -28639.476} C_VEL
LIN {X 0,Y 108.685,Z 357.327,A -85,B 0,C 180,E1 -28643.393,E2 -28643.393} C_VEL
LIN {X 0,Y 111.504,Z 363.248,A -85,B 0,C 180,E1 -28647.447,E2 -28647.447} C_VEL
LIN {X 0,Y 112.794,Z 366.526,A -85,B 0,C 180,E1 -28649.301,E2 -28649.301} C_VEL
LIN {X 0,Y 111.461,Z 375.065,A -85,B 0,C 180,E1 -28649.983,E2 -28649.983} C_VEL
LIN {X 0,Y 109.597,Z 383.161,A -85,B 0,C 180,E1 -28650.865,E2 -28650.865} C_VEL
LIN {X 0,Y 108.607,Z 386.905,A -85,B 0,C 180,E1 -28651.392,E2 -28651.392} C_VEL
LIN {X 0,Y 107.176,Z 390.616,A -85,B 0,C 180,E1 -28651.605,E2 -28651.605} C_VEL
LIN {X 0,Y 103.635,Z 396.348,A -85,B 0,C 180,E1 -28651.132,E2 -28651.132} C_VEL
LIN {X 0,Y 99.683,Z 401.825,A -85,B 0,C 180,E1 -28650.769,E2 -28650.769} C_VEL
LIN {X 0,Y 97.593,Z 405.134,A -85,B 0,C 180,E1 -28651.224,E2 -28651.224} C_VEL
LIN {X 0,Y 92.103,Z 414.452,A -85,B 0,C 180,E1 -28653.916,E2 -28653.916} C_VEL
LIN {X 0,Y 87.429,Z 421.121,A -85,B 0,C 180,E1 -28656.497,E2 -28656.497} C_VEL
LIN {X 0,Y 82.363,Z 427.43,A -85,B 0,C 180,E1 -28659.825,E2 -28659.825} C_VEL
LIN {X 0,Y 77.501,Z 432.677,A -85,B 0,C 180,E1 -28663.489,E2 -28663.489} C_VEL
LIN {X 0,Y 73.002,Z 437.051,A -85,B 0,C 180,E1 -28667.628,E2 -28667.628} C_VEL
LIN {X 0,Y 66.943,Z 442.199,A -85,B 0,C 180,E1 -28674.727,E2 -28674.727} C_VEL
LIN {X 0,Y 63.566,Z 444.831,A -85,B 0,C 180,E1 -28680.159,E2 -28680.159} C_VEL
LIN {X 0,Y 59.647,Z 447.707,A -85,B 0,C 180,E1 -28689.296,E2 -28689.296} C_VEL
LIN {X 0,Y 57.764,Z 448.962,A -85,B 0,C 180,E1 -28695.913,E2 -28695.913} C_VEL
LIN {X 0,Y 56.626,Z 449.75,A -85,B 0,C 180,E1 -28702.867,E2 -28702.867} C_VEL
LIN {X 0,Y 56.225,Z 450.051,A -85,B 0,C 180,E1 -28709.996,E2 -28709.996} C_VEL
LIN {X 0,Y 56.625,Z 449.768,A -85,B 0,C 180,E1 -28717.126,E2 -28717.126} C_VEL
LIN {X 0,Y 57.762,Z 449.017,A -85,B 0,C 180,E1 -28724.08,E2 -28724.08} C_VEL
LIN {X 0,Y 59.605,Z 447.802,A -85,B 0,C 180,E1 -28730.712,E2 -28730.712} C_VEL
LIN {X 0,Y 63.551,Z 444.962,A -85,B 0,C 180,E1 -28739.84,E2 -28739.84} C_VEL
LIN {X 0,Y 66.92,Z 442.371,A -85,B 0,C 180,E1 -28745.279,E2 -28745.279} C_VEL
LIN {X 0,Y 72.953,Z 437.273,A -85,B 0,C 180,E1 -28752.399,E2 -28752.399} C_VEL
LIN {X 0,Y 78.639,Z 431.784,A -85,B 0,C 180,E1 -28757.498,E2 -28757.498} C_VEL
LIN {X 0,Y 84.848,Z 424.872,A -85,B 0,C 180,E1 -28761.891,E2 -28761.891} C_VEL
LIN {X 0,Y 90.685,Z 416.941,A -85,B 0,C 180,E1 -28765.425,E2 -28765.425} C_VEL
LIN {X 0,Y 95.471,Z 409.368,A -85,B 0,C 180,E1 -28767.835,E2 -28767.835} C_VEL
LIN {X 0,Y 99.033,Z 402.908,A -85,B 0,C 180,E1 -28769.364,E2 -28769.364} C_VEL
LIN {X 0,Y 102.564,Z 395.058,A -85,B 0,C 180,E1 -28770.883,E2 -28770.883} C_VEL
LIN {X 0,Y 105.472,Z 386.904,A -85,B 0,C 180,E1 -28772.136,E2 -28772.136} C_VEL
LIN {X 0,Y 108.13,Z 376.741,A -85,B 0,C 180,E1 -28773.292,E2 -28773.292} C_VEL
LIN {X 0,Y 109.363,Z 370.091,A -85,B 0,C 180,E1 -28773.904,E2 -28773.904} C_VEL
LIN {X 0,Y 106.991,Z 363.786,A -85,B 0,C 180,E1 -28778.22,E2 -28778.22} C_VEL
LIN {X 0,Y 104.542,Z 358.66,A -85,B 0,C 180,E1 -28783.147,E2 -28783.147} C_VEL
LIN {X 0,Y 102.741,Z 355.045,A -85,B 0,C 180,E1 -28788.157,E2 -28788.157} C_VEL
LIN {X 0,Y 101.399,Z 351.913,A -85,B 0,C 180,E1 -28795.029,E2 -28795.029} C_VEL
LIN {X 0,Y 101.305,Z 350.871,A -85,B 0,C 180,E1 -28797.017,E2 -28797.017} C_VEL
LIN {X 0,Y 101.289,Z 350.84,A -85,B 0,C 180,E1 -28801.988,E2 -28801.988} C_VEL
LIN {X 0,Y 102.734,Z 355.051,A -85,B 0,C 180,E1 -28811.093,E2 -28811.093} C_VEL
LIN {X 0,Y 104.898,Z 359.467,A -85,B 0,C 180,E1 -28816.95,E2 -28816.95} C_VEL
LIN {X 0,Y 107.079,Z 363.991,A -85,B 0,C 180,E1 -28821.192,E2 -28821.192} C_VEL
LIN {X 0,Y 108.237,Z 366.996,A -85,B 0,C 180,E1 -28823.187,E2 -28823.187} C_VEL
LIN {X 0,Y 109.317,Z 371.94,A -85,B 0,C 180,E1 -28825.397,E2 -28825.397} C_VEL
LIN {X 0,Y 107.685,Z 381.046,A -85,B 0,C 180,E1 -28825.965,E2 -28825.965} C_VEL
LIN {X 0,Y 105.088,Z 390.688,A -85,B 0,C 180,E1 -28826.835,E2 -28826.835} C_VEL
LIN {X 0,Y 101.507,Z 400.365,A -85,B 0,C 180,E1 -28828.027,E2 -28828.027} C_VEL
LIN {X 0,Y 96.318,Z 411.088,A -85,B 0,C 180,E1 -28829.953,E2 -28829.953} C_VEL
LIN {X 0,Y 91.29,Z 419.356,A -85,B 0,C 180,E1 -28832.136,E2 -28832.136} C_VEL
LIN {X 0,Y 85.737,Z 427.042,A -85,B 0,C 180,E1 -28834.949,E2 -28834.949} C_VEL
LIN {X 0,Y 80.473,Z 433.378,A -85,B 0,C 180,E1 -28838.191,E2 -28838.191} C_VEL
LIN {X 0,Y 75.491,Z 438.645,A -85,B 0,C 180,E1 -28841.865,E2 -28841.865} C_VEL
LIN {X 0,Y 70.891,Z 443.043,A -85,B 0,C 180,E1 -28846.059,E2 -28846.059} C_VEL
LIN {X 0,Y 64.834,Z 448.243,A -85,B 0,C 180,E1 -28853.406,E2 -28853.406} C_VEL
LIN {X 0,Y 61.506,Z 450.904,A -85,B 0,C 180,E1 -28859.06,E2 -28859.06} C_VEL
LIN {X 0,Y 57.913,Z 453.848,A -85,B 0,C 180,E1 -28868.654,E2 -28868.654} C_VEL
LIN {X 0,Y 56.445,Z 455.123,A -85,B 0,C 180,E1 -28875.584,E2 -28875.584} C_VEL
LIN {X 0,Y 55.783,Z 455.924,A -85,B 0,C 180,E1 -28882.766,E2 -28882.766} C_VEL
LIN {X 0,Y 55.893,Z 456.241,A -85,B 0,C 180,E1 -28890.004,E2 -28890.004} C_VEL
LIN {X 0,Y 55.785,Z 455.909,A -85,B 0,C 180,E1 -28897.241,E2 -28897.241} C_VEL
LIN {X 0,Y 56.446,Z 455.08,A -85,B 0,C 180,E1 -28904.423,E2 -28904.423} C_VEL
LIN {X 0,Y 57.914,Z 453.776,A -85,B 0,C 180,E1 -28911.353,E2 -28911.353} C_VEL
LIN {X 0,Y 61.507,Z 450.801,A -85,B 0,C 180,E1 -28920.947,E2 -28920.947} C_VEL
LIN {X 0,Y 64.836,Z 448.108,A -85,B 0,C 180,E1 -28926.6,E2 -28926.6} C_VEL
LIN {X 0,Y 70.888,Z 442.869,A -85,B 0,C 180,E1 -28933.951,E2 -28933.951} C_VEL
LIN {X 0,Y 76.729,Z 437.25,A -85,B 0,C 180,E1 -28939.087,E2 -28939.087} C_VEL
LIN {X 0,Y 83.684,Z 429.36,A -85,B 0,C 180,E1 -28943.873,E2 -28943.873} C_VEL
LIN {X 0,Y 89.199,Z 422.07,A -85,B 0,C 180,E1 -28946.844,E2 -28946.844} C_VEL
LIN {X 0,Y 94.118,Z 414.344,A -85,B 0,C 180,E1 -28949.178,E2 -28949.178} C_VEL
LIN {X 0,Y 98.499,Z 406.23,A -85,B 0,C 180,E1 -28950.936,E2 -28950.936} C_VEL
LIN {X 0,Y 102.243,Z 397.813,A -85,B 0,C 180,E1 -28952.256,E2 -28952.256} C_VEL
LIN {X 0,Y 105.313,Z 389.179,A -85,B 0,C 180,E1 -28953.212,E2 -28953.212} C_VEL
LIN {X 0,Y 108.029,Z 378.329,A -85,B 0,C 180,E1 -28954.153,E2 -28954.153} C_VEL
LIN {X 0,Y 109.052,Z 371.906,A -85,B 0,C 180,E1 -28954.523,E2 -28954.523} C_VEL
LIN {X 0,Y 107.863,Z 366.156,A -85,B 0,C 180,E1 -28956.987,E2 -28956.987} C_VEL
LIN {X 0,Y 105.615,Z 361.237,A -85,B 0,C 180,E1 -28960.945,E2 -28960.945} C_VEL
LIN {X 0,Y 103.949,Z 357.95,A -85,B 0,C 180,E1 -28964.53,E2 -28964.53} C_VEL
LIN {X 0,Y 102.513,Z 354.913,A -85,B 0,C 180,E1 -28968.633,E2 -28968.633} C_VEL
LIN {X 0,Y 101.169,Z 351.841,A -85,B 0,C 180,E1 -28975.081,E2 -28975.081} C_VEL
LIN {X 0,Y 101.036,Z 350.81,A -85,B 0,C 180,E1 -28977.01,E2 -28977.01} C_VEL
LIN {X 0,Y 100.914,Z 350.667,A -85,B 0,C 180,E1 -28981.996,E2 -28981.996} C_VEL
LIN {X 0,Y 101.072,Z 351.152,A -85,B 0,C 180,E1 -28984.487,E2 -28984.487} C_VEL
LIN {X 0,Y 102.158,Z 354.467,A -85,B 0,C 180,E1 -28991.027,E2 -28991.027} C_VEL
LIN {X 0,Y 102.738,Z 355.376,A -85,B 0,C 180,E1 -28992.924,E2 -28992.924} C_VEL
LIN {X 0,Y 104.775,Z 359.566,A -85,B 0,C 180,E1 -28998.168,E2 -28998.168} C_VEL
LIN {X 0,Y 106.926,Z 363.973,A -85,B 0,C 180,E1 -29002.288,E2 -29002.288} C_VEL
LIN {X 0,Y 109.128,Z 369.83,A -85,B 0,C 180,E1 -29006.254,E2 -29006.254} C_VEL
LIN {X 0,Y 106.798,Z 381.224,A -85,B 0,C 180,E1 -29007.27,E2 -29007.27} C_VEL
LIN {X 0,Y 104.02,Z 390.487,A -85,B 0,C 180,E1 -29008.555,E2 -29008.555} C_VEL
LIN {X 0,Y 100.494,Z 399.243,A -85,B 0,C 180,E1 -29010.063,E2 -29010.063} C_VEL
LIN {X 0,Y 97.593,Z 405.134,A -85,B 0,C 180,E1 -29011.224,E2 -29011.224} C_VEL
LIN {X 0,Y 94.535,Z 410.091,A -85,B 0,C 180,E1 -29012.22,E2 -29012.22} C_VEL
LIN {X 0,Y 88.219,Z 417.583,A -85,B 0,C 180,E1 -29013.113,E2 -29013.113} C_VEL
LIN {X 0,Y 81.404,Z 424.467,A -85,B 0,C 180,E1 -29014.374,E2 -29014.374} C_VEL
LIN {X 0,Y 77.628,Z 428.233,A -85,B 0,C 180,E1 -29016.073,E2 -29016.073} C_VEL
LIN {X 0,Y 71.561,Z 434.234,A -85,B 0,C 180,E1 -29020.432,E2 -29020.432} C_VEL
LIN {X 0,Y 65.6,Z 439.344,A -85,B 0,C 180,E1 -29025.859,E2 -29025.859} C_VEL
LIN {X 0,Y 59.363,Z 444.06,A -85,B 0,C 180,E1 -29033.7,E2 -29033.7} C_VEL
LIN {X 0,Y 55.882,Z 446.36,A -85,B 0,C 180,E1 -29039.793,E2 -29039.793} C_VEL
LIN {X 0,Y 53.082,Z 448.099,A -85,B 0,C 180,E1 -29046.593,E2 -29046.593} C_VEL
LIN {X 0,Y 50.926,Z 449.353,A -85,B 0,C 180,E1 -29053.974,E2 -29053.974} C_VEL
LIN {X 0,Y 49.614,Z 450.14,A -85,B 0,C 180,E1 -29061.852,E2 -29061.852} C_VEL
LIN {X 0,Y 49.16,Z 450.441,A -85,B 0,C 180,E1 -29069.996,E2 -29069.996} C_VEL
LIN {X 0,Y 49.612,Z 450.158,A -85,B 0,C 180,E1 -29078.14,E2 -29078.14} C_VEL
LIN {X 0,Y 50.923,Z 449.408,A -85,B 0,C 180,E1 -29086.019,E2 -29086.019} C_VEL
LIN {X 0,Y 53.028,Z 448.193,A -85,B 0,C 180,E1 -29093.424,E2 -29093.424} C_VEL
LIN {X 0,Y 57.52,Z 445.352,A -85,B 0,C 180,E1 -29103.351,E2 -29103.351} C_VEL
LIN {X 0,Y 61.276,Z 442.761,A -85,B 0,C 180,E1 -29109.106,E2 -29109.106} C_VEL
LIN {X 0,Y 67.882,Z 437.663,A -85,B 0,C 180,E1 -29116.442,E2 -29116.442} C_VEL
LIN {X 0,Y 74.031,Z 432.174,A -85,B 0,C 180,E1 -29121.55,E2 -29121.55} C_VEL
LIN {X 0,Y 80.671,Z 425.26,A -85,B 0,C 180,E1 -29125.852,E2 -29125.852} C_VEL
LIN {X 0,Y 86.869,Z 417.328,A -85,B 0,C 180,E1 -29129.266,E2 -29129.266} C_VEL
LIN {X 0,Y 91.9,Z 409.754,A -85,B 0,C 180,E1 -29131.572,E2 -29131.572} C_VEL
LIN {X 0,Y 95.613,Z 403.295,A -85,B 0,C 180,E1 -29133.025,E2 -29133.025} C_VEL
LIN {X 0,Y 99.31,Z 395.443,A -85,B 0,C 180,E1 -29134.456,E2 -29134.456} C_VEL
LIN {X 0,Y 102.991,Z 385.253,A -85,B 0,C 180,E1 -29135.86,E2 -29135.86} C_VEL
LIN {X 0,Y 105.433,Z 375.805,A -85,B 0,C 180,E1 -29136.849,E2 -29136.849} C_VEL
LIN {X 0,Y 105.888,Z 373.406,A -85,B 0,C 180,E1 -29137.154,E2 -29137.154} C_VEL
LIN {X 0,Y 104.186,Z 368.262,A -85,B 0,C 180,E1 -29141.248,E2 -29141.248} C_VEL
LIN {X 0,Y 102.689,Z 364.61,A -85,B 0,C 180,E1 -29145.321,E2 -29145.321} C_VEL
LIN {X 0,Y 101.431,Z 361.661,A -85,B 0,C 180,E1 -29149.583,E2 -29149.583} C_VEL
